(* Logix 5000 project; controller DC01 vendor 1 type 14 code 165 rev 32.12; software revision 32.04 *)

TASK MainTask (continuous, watchdog 500 ms) : MainProgram, LN01, LN02, LN03, LN04

MODULES
   Local : vendor 1 type 14 code 165 (ICP 0, rev 32.12)
      ASSY_LN01 : 1756-EN2T (ICP 1, Ethernet 192.168.1.211, rev 11.1)
         LN01_COMMS : 1756-EN2T (Ethernet 192.168.1.221, rev 11.2, Output RPI 10 ms)
            LN01 : vendor 1 type 14 code 167 (ICP 0, rev 32.1)
      ASSY_LN02 : 1756-EN2T (ICP 2, Ethernet 192.168.1.212, rev 11.1)
         LN02_COMMS : 1756-EN2T (Ethernet 192.168.1.222, rev 11.1, Output RPI 10 ms)
            LN02 : vendor 1 type 14 code 167 (ICP 0, rev 33.1)
      ASSY_LN03 : 1756-EN2T (ICP 3, Ethernet 192.168.1.213, rev 11.1)
         LN03_COMMS : 1756-EN2T (Ethernet 192.168.1.223, rev 11.1, Output RPI 10 ms)
            LN03 : vendor 1 type 14 code 167 (ICP 0, rev 33.1)
      ASSY_COMMS : 1756-EN2T (ICP 6, Ethernet 10.27.36.150, rev 11.2)
      ASSY_LN04 : 1756-EN2T (ICP 4, Ethernet 192.168.1.214, rev 11.1)
         LN04_COMMS : 1756-EN2T (Ethernet 192.168.1.224, rev 11.1, Output RPI 10 ms)
            LN04 : vendor 1 type 14 code 167 (ICP 0, rev 33.1)
END_MODULES

TYPE Barcode_SNModel :
STRUCT
   Data : STRING[5];
   Bit : BOOL[32];
END_STRUCT
END_TYPE

TYPE BARCODESCAN :
STRUCT
   RAWDATA : STRING;
   TRIGGER : BOOL;
   CLEAR : BOOL;
   SCANCOMPLETE : BOOL;
END_STRUCT
END_TYPE

TYPE Data_RECT :
STRUCT
   Volt_Out : INT;
   Amp_Out : INT;
   DC_ON : BOOL;
END_STRUCT
END_TYPE

TYPE DateTime_Type :   // Structure for the DateTime from the Controller wallclock accessed by the GSV/SSV instruction
STRUCT
   Year : DINT;
   Month : DINT;   // The month (1 - 12)
   Day : DINT;   // The day (1 - 31)
   Hour : DINT;   // hour (0 - 23)
   Minute : DINT;   // minute (0 - 59)
   Second : DINT;   // second (0 - 59)
   Microseconds : DINT;   // (0 - 999,999)
END_STRUCT
END_TYPE

TYPE DriveData :
STRUCT
   FieldAmps : REAL;
   VoltsOut : REAL;
   ArmCurrent : REAL;
   ActualSpeed : REAL;
END_STRUCT
END_TYPE

TYPE DriveDataDINT :
STRUCT
   FieldAmps : DINT;
   ArmAmps : DINT;
   OutVolts : DINT;
   Speed : DINT;
END_STRUCT
END_TYPE

TYPE Drives1079 :
STRUCT
   Drive1 : DriveData;
   Drive2 : DriveData;
   Drive3 : DriveData;
   Drive4 : DriveData;
   Drive5 : DriveData;
   Drive6 : DriveData;
END_STRUCT
END_TYPE

TYPE Drives1079DINT :
STRUCT
   Drive1 : DriveDataDINT;
   Drive2 : DriveDataDINT;
   Drive3 : DriveDataDINT;
   Drive4 : DriveDataDINT;
   Drive5 : DriveDataDINT;
   Drive6 : DriveDataDINT;
END_STRUCT
END_TYPE

TYPE Lodestar_Data_DINTS :
STRUCT
   Mode : DINT;
   State : DINT;
   AutoMan : DINT;
   Process : DINT;
   Rate : DINT;
   Fault_Code : DINT;
   Infeed_Count : DINT;
   OutFeed_Count : DINT;
   Reject_Count : DINT;
   Cycle_Count : DINT;
END_STRUCT
END_TYPE

TYPE LPNSTATUS :   // Data From SQL for Online Printing to tell what Current Model the line is in
STRUCT
   LineID : INT;   // Line Number
   Total_Run : INT;   // Total Number of Units in Current Run
   Produced : INT;   // Total Number of Units Ran in Current Run
   Left_To_Run : INT;   // Total Number of Units Left to Run in Current Run
   Model : STRING;   // Model Number of Current Run
END_STRUCT
END_TYPE

TYPE OnlinePrinitng :
STRUCT
   ENGMODEL : STRING;
   SALESMODEL : STRING;
   MODEL : STRING;
   SERIAL : STRING;
   DATA_TO_APP_READY : BOOL;
   APP_DATA_RECEIVED : BOOL;
   DATA_FROM_APP_READY : BOOL;
   LINERUNNING : BOOL;
   CLEAR : BOOL;
   BARCODEDATA : BARCODESCAN;
END_STRUCT
END_TYPE

TYPE PA_WallClock_UDDT :
STRUCT
   One_Shots : BOOL[128];
   Bool : BOOL[128];
   Real : REAL[50];
   Dbl_Int : DINT[50];
   Int : INT[50];
   Pointer1 : INT;
   Pointer2 : INT;
   Pointer3 : INT;
   Pointer4 : INT;
   Pointer5 : INT;
   Timer : TIMER[50];
   Counter : COUNTER[25];
   Control : CONTROL[16];
END_STRUCT
END_TYPE

TYPE R1_Lines_Status_to_R2 :
STRUCT
   LN02 : UDT_Line_Status_to_R2;
   LN03 : UDT_Line_Status_to_R2;
   LN04 : UDT_Line_Status_to_R2;
   LN07 : UDT_Line_Status_to_R2;
END_STRUCT
END_TYPE

TYPE R3_Ticket_Data :   // Ticket Data from LN04 Scanners
STRUCT
   Model : STRING;
   Date : STRING;
   Serial : STRING;
END_STRUCT
END_TYPE

TYPE R3_Ticket_Data2 :
STRUCT
   Model : STRING;
   Date : STRING;
   Serial : STRING;
END_STRUCT
END_TYPE

TYPE RECT_1079 :
STRUCT
   RECT1 : Data_RECT;
   RECT2 : Data_RECT;
   RECTBU : Data_RECT;
END_STRUCT
END_TYPE

TYPE STRING_12 :
STRUCT
   LEN : DINT;
   DATA : SINT[12];
END_STRUCT
END_TYPE

TYPE STRING_16 :
STRUCT
   LEN : DINT;
   DATA : SINT[16];
END_STRUCT
END_TYPE

TYPE STRING_24 :
STRUCT
   LEN : DINT;
   DATA : SINT[24];
END_STRUCT
END_TYPE

TYPE STRING_4 :
STRUCT
   LEN : DINT;
   DATA : SINT[4];
END_STRUCT
END_TYPE

TYPE STRING_40 :
STRUCT
   LEN : DINT;
   DATA : SINT[40];
END_STRUCT
END_TYPE

TYPE UDT_Current_Status :
STRUCT
   Area : STRING_12;
   Line : STRING_12;
   Shift : DINT;
   _1st_Shift_Avail : BOOL;
   _1st_Shift_Active : BOOL;
   _1st_Shift_Scheduled : BOOL;
   _2nd_Shift_Avail : BOOL;
   _2nd_Shift_Active : BOOL;
   _2nd_Shift_Scheduled : BOOL;
   _3rd_Shift_Avail : BOOL;
   _3rd_Shift_Active : BOOL;
   _3rd_Shift_Scheduled : BOOL;
   DayOfWeek : STRING_16;
   DayOfWeek_Int : DINT;
   Start_Time : STRING_16;
   End_Time : STRING_16;
   _1st_Break_Time : STRING_16;
   _1st_Break_Trigger : BOOL;
   _1st_Break_Active : BOOL;
   _1st_Break_Used : BOOL;
   Lunch_Time : STRING_16;
   Lunch_Trigger : BOOL;
   Lunch_Active : BOOL;
   Lunch_Used : BOOL;
   _2nd_Break_Time : STRING_16;
   _2nd_Break_Trigger : BOOL;
   _2nd_Break_Active : BOOL;
   _2nd_Break_Used : BOOL;
   Rotate_Active : BOOL;
   Rotate_Cmd : BOOL;   // 30 Second Downtime Event to Rotate the Crew
   Scheduled_Units : DINT;
   Line_Rate : DINT;   // Seconds to Construct a Component
   Line_Rate_SP : REAL;
   Units_Remaining : DINT;
   Units_Produced : DINT;
   Units_Scrapped : DINT;
   Units_Lossed : DINT;
   AY_Percent : REAL;
   Shift_Minutes_Remainng : DINT;
   Shift_Seconds_Remaining : DINT;
   DownTime_Code : DINT;
   Flex_Cmd : BOOL;
   Flex_Active : BOOL;
   FlexTo_Line : STRING_16;
   Flex_EndCmd : BOOL;
   Rotate_LEN : REAL;   // seconds
   Brk_LEN : REAL;   // minutes
   Lunch_LEN : REAL;   // minutes
   Break_Stop_On : BOOL;
   Break_Stop_Allowed : BOOL;
   Flex_Stop_On : BOOL;
   Flex_Stop_Allowed : BOOL;
   Rotate_Stop_On : BOOL;
   Rotate_Stop_Allowed : BOOL;
   S1_Scheduled : DINT;
   S2_Scheduled : DINT;
   S3_Scheduled : DINT;
   Shift_Scheduled : BOOL;
   Shift_Active : BOOL;
   RateToMakeSchedule : REAL;
   Theoretical_Units : DINT;
   Standard_LineRate : REAL;
   Running : BOOL;
   State : DINT;
   LineWide_Event : DINT;
   Units_Rejected : DINT;
END_STRUCT
END_TYPE

TYPE UDT_Daily_Schedule :
STRUCT
   _1st_Shift_Avail : BOOL;
   _1st_Shift_Start : STRING_16;
   _1st_Shift_End : STRING_16;
   _1st_Shift_Break1_Start : STRING_16;
   _1st_Shift_Break1_Length : DINT;   // Minutes
   _1st_Shift_Lunch_Start : STRING_16;
   _1st_Shift_Lunch_Length : DINT;   // Minutes
   _1st_Shift_Break2_Start : STRING_16;
   _1st_Shift_Break2_Length : DINT;   // Minutes
   _2nd_Shift_Avail : BOOL;
   _2nd_Shift_Start : STRING_16;
   _2nd_Shift_End : STRING_16;
   _2nd_Shift_Break1_Start : STRING_16;
   _2nd_Shift_Break1_Length : DINT;   // Minutes
   _2nd_Shift_Lunch_Start : STRING_16;
   _2nd_Shift_Lunch_Length : DINT;   // Minutes
   _2nd_Shift_Break2_Start : STRING_16;
   _2nd_Shift_Break2_Length : DINT;   // Minutes
   _3rd_Shift_Avail : BOOL;
   _3rd_Shift_Start : STRING_16;
   _3rd_Shift_End : STRING_16;
   _3rd_Shift_Break1_Start : STRING_16;
   _3rd_Shift_Break1_Length : DINT;   // Minutes
   _3rd_Shift_Lunch_Start : STRING_16;
   _3rd_Shift_Lunch_Length : DINT;   // Minutes
   _3rd_Shift_Break2_Start : STRING_16;
   _3rd_Shift_Break2_Length : DINT;   // Minutes
   Rotate_Length : DINT;   // Seconds
   Break_Stop_On : BOOL;
   Break_Stop_Allowed : BOOL;
   Flex_Stop_On : BOOL;
   Flex_Stop_Allowed : BOOL;
   Rotate_Stop_On : BOOL;
   Rotate_Stop_Allowed : BOOL;
   S1_Scheduled : DINT;
   S2_Scheduled : DINT;
   S3_Scheduled : DINT;
   RateToMakeSchedule : REAL;
END_STRUCT
END_TYPE

TYPE UDT_DateTime :
STRUCT
   Year : STRING_4;
   Month : STRING_4;
   Day : STRING_4;
   Hour : STRING_4;
   Minute : STRING_4;
   Second : STRING_4;
   MicroSecond : STRING_4;
   ForwardSlash : STRING_4;
   Colon : STRING_4;
   Period : STRING_4;
   Zero : STRING_4;
   Final : STRING_4;
   Space : STRING_4;
   Millisecond : STRING_4;
END_STRUCT
END_TYPE

TYPE UDT_Downtime_Testing :
STRUCT
   Line_Scheduled : BOOL;
   Break : BOOL;
   Set_ModelNumber : BOOL;
   Downtime_Active : BOOL;
   Shift_Reset : BOOL;
   CrateCount_Trigger : BOOL;
   Set_TAKT : BOOL;
   TAKT_Time : DINT;
   SerialNumber_Length : DINT;
   Dev : DINT;
   Current_Shift : DINT;
   OneShots : DINT;
   LineRate : REAL;
   Production_Crate_Count_TMR : TIMER;
   Set_TAKT_Delay_TMR : TIMER;
   CrateCountTrigger_TMR : TIMER;
   Sch_Production_Crate_Count_TMR : TIMER;
   SerialNumber_Generator_CNTR : COUNTER;
   Units_Produced_CNTR : COUNTER;
   Scheduled_Units_CNTR : COUNTER;
   ModelNumber : STRING;
   TempModelNumber : STRING;
   SerialNumber : STRING;
   SalesModelNumber : STRING;
   zeros_7 : STRING_12;
   zeros_6 : STRING_12;
   zeros_5 : STRING_12;
   zeros_4 : STRING_12;
   zeros_3 : STRING_4;
   zeros_2 : STRING_4;
   zeros_1 : STRING_4;
   LineID : STRING;
END_STRUCT
END_TYPE

TYPE UDT_Line_Status_to_R2 :
STRUCT
   Active_Shift : DINT;
   Count : DINT;
   Break_Active : BOOL;
   DT_Active : BOOL;
END_STRUCT
END_TYPE

TYPE UDT_R3_BlackOut :   // Defines start and stop times for R3 schedule true ups, this apples to all lines in Clyde
STRUCT
   Starthour : DINT;
   StartMinute : DINT;
   EndHour : DINT;
   EndMinute : DINT;
END_STRUCT
END_TYPE

TYPE UDT_R3_Missed_Scan :
STRUCT
   New_Serial : BOOL;
   Same_Serial_TMR : TIMER;
   Prev_Count : DINT;
   New_Serial_TMR : TIMER;
   Missed_Scan_TMR : TIMER;
   Prev_Serial : STRING;
END_STRUCT
END_TYPE

TYPE UDT_R3_Model_Information :   // Provides structure for getting information from Ignition related to Changeover information
STRUCT
   Model : STRING;
   Count : DINT;
   Order : DINT;
   SEQ_No : DINT;
   SAP_Received_QTY : DINT;
   Description : STRING;
END_STRUCT
END_TYPE

TYPE UDT_ScantoExitDatatoDC :
STRUCT
   Serial : STRING;
   Model : STRING;
   Pass : BOOL;
   Fail : BOOL;
   Location : DINT;
END_STRUCT
END_TYPE

TYPE UDT_SHIFT_FPY :   // Shift FPY FOR line 2,3,4,7
STRUCT
   Line_2_FPY : REAL;   // Line 2
   Line_3_FPY : REAL;   // Line 3
   Line_4_FPY : REAL;   // Line 4
   Line_7_FPY : REAL;   // Line 7
END_STRUCT
END_TYPE

TYPE UDT_ShiftString_Breakdown :
STRUCT
   s1StartHour : STRING_4;
   s1StartMin : STRING_4;
   s1EndHour : STRING_4;
   s1_EndMin : STRING_4;
   s2StartHour : STRING_4;
   s2StartMin : STRING_4;
   s2EndHour : STRING_4;
   s2EndMin : STRING_4;
   s3StartHour : STRING_4;
   s3StartMin : STRING_4;
   s3EndHour : STRING_4;
   s3EndMin : STRING_4;
   break1StartHour : STRING_4;
   break1StartMin : STRING_4;
   break2StartHour : STRING_4;
   break2StartMin : STRING_4;
   lunchStartHour : STRING_4;
   lunchStartMin : STRING_4;
END_STRUCT
END_TYPE

TYPE udt_SKU :
STRUCT
   Name : STRING;   // Name of product
   Diameter : REAL;   // Diameter in millimeters
   Height : REAL;   // Height in millimeters
   ID : INT;   // Product ID
   DiameterID : REAL;
   HeightID : REAL;
   Update : BOOL;
   Update_ONS : BOOL;
   Active : BOOL;
   Active_Req : BOOL;
   UpdatePB : BOOL;
   TooManyActive : BOOL;
   DestinationOut : INT;
   ActivePB : BOOL;
   BatchRequest : INT;
   BatchCount : INT;
   ASRS_Enabled : BOOL;
   DestinationIn : INT;
   ResetPB : BOOL;
   BatchComplete : BOOL;
END_STRUCT
END_TYPE

TYPE UDT_SN_Model :
STRUCT
   writeIndex : DINT;
   readIndex : DINT;
   LastReadCode : DINT;
   Serial : STRING_16;
   Model : STRING_16;
   DateTime : STRING_24;
   newData : BOOL;
END_STRUCT
END_TYPE

TYPE UDT_Visual_Inspect_Data :   // UDT from Assy lines for Scanners that track models
STRUCT
   Date : STRING;
   Unit_Status : BOOL;
   Model : STRING;
   Serial : STRING;
   Badge_ID : DINT;
   Data_Ready : BOOL;
END_STRUCT
END_TYPE

TYPE UDT_Visual_Inspect_Data2 :
STRUCT
   DATE : STRING;
   UNIT_STATUS : BOOL;
   MODEL : STRING;
   SERIAL : STRING;
   BADGE_ID : DINT;
   DATA_READY : BOOL;
END_STRUCT
END_TYPE

TYPE UDT_Weekly_Schedule :
STRUCT
   Monday : UDT_Daily_Schedule;
   Tuesday : UDT_Daily_Schedule;
   Wednesday : UDT_Daily_Schedule;
   Thursday : UDT_Daily_Schedule;
   Friday : UDT_Daily_Schedule;
   Saturday : UDT_Daily_Schedule;
   Sunday : UDT_Daily_Schedule;
END_STRUCT
END_TYPE

TYPE Visual_Inspect_Data :
STRUCT
   DATE : STRING;
   UNIT_STATUS : BOOL;
   MODEL : STRING;
   SERIAL : STRING;
   BADGE_ID : DINT;
   DATA_READY : BOOL;
END_STRUCT
END_TYPE

VAR_GLOBAL   (* controller tags *)
   Always_Off : BOOL;
   apc_debounce : TIMER := (PRE := 1100);
   apc_DT_CTR : TIMER := (PRE := 999999999);
   ASSY_COMS_com_status : DINT := 16384;   // DC01 Bldg Ethernet Communications To Data Center Status Monitor
   ay : REAL := 0.8867925;
   ay_LN01 : DINT;
   ay_LN01_REAL : REAL := 0.95028526;
   AY_LN02_REAL : REAL := 0.9279279;
   Barcode_Scan : MESSAGE;
        MessageParameters(ServiceCode := 16#004c, LocalElement := LN01_Messages_Barcode_SNModel, ...)
   brentest : BOOL;
   brentest2 : BOOL := 1;
   Brian_Test : BOOL;
   ChangeWEM15TO12 : BOOL := 1;
   clock_current_string : STRING[13] := ([0] := '2023', [1] := '5', [2] := '8', [3] := '7', [4] := '52', [5] := '42');
   Clock_Min_Pulse : BOOL;
   Clock_Set_Routine : PA_WallClock_UDDT := (Bool[20] := 1, Dbl_Int[40] := 2023, Dbl_Int[41] := 5, Dbl_Int[42] := 8, Dbl_Int[43] := 7, Dbl_Int[44] := 52, Dbl_Int[45] := 43, Dbl_Int[46] := 547971, Timer[0].PRE := 500, Timer[8].EN := 1, Timer[8].TT := 1, Timer[9].ACC := 100, Timer[9].EN := 1, Timer[9].DN := 1);
   covid19 : BOOL;
   CurrentSchedule : UDT_ShiftString_Breakdown := (s1StartHour := '20', s1StartMin := '3-', s1EndHour := '20', s1_EndMin := '3-', s2StartHour := '20', s2StartMin := '3-', s2EndHour := '20', s2EndMin := '3-', s3StartHour := '20', s3StartMin := '3-', s3EndHour := '20', s3EndMin := '3-');
   DateTime_Update : BOOL;
   DayOfWeek : DINT;
   DC01_to_LN04_Data : DINT[26] := ([1] := 201);
   DC1_clock_sync : DINT[10] := ([0] := 2023, [1] := 5, [2] := 8, [3] := 7, [4] := 52, [5] := 43);
   DC1_OPCFault : BOOL := 1;
   DC1_OPCWatchDog : BOOL := 1;
   DC1_to_LN01_Messages : DINT[20] := ([0] := 1, [2] := 1, [3] := 1240, [4] := 598, [5] := 7, [6] := 5, [7] := 15, [8] := 28, [9] := 15, [10] := 35, [11] := 23, [12] := 58, [14] := 5, [15] := 6, [16] := 58, [17] := 33900, [19] := 1);
        [10]   // CURRENT SCHEDULE SHIFT 2 START MINUTE
        [11]   // CURRENT SCHEDULE SHIFT 2 END HOUR
        [12]   // CURRENT SCHEDULE SHIFT 2 END MINUTE
        [13]   // CURRENT SCHEDULE SHIFT 3 START HOUR
        [14]   // CURRENT SCHEDULE SHIFT 3 START MINUTE
        [15]   // CURRENT SCHEDULE SHIFT 3 END HOUR
        [16]   // CURRENT SCHEDULE SHIFT 3 END MINUTE
        [17]   // CURRENT SCHEDULE AVAILABLE SECONDS
        [19].0   // SHIFT SCHEDULED
        [19].1   // OPC COMMS OKAY
        [2]   // ACTIVE SHIFT
        [3]   // SCHEDULED UNITS
        [5]   // CURRENT SCHEDULE SHIFT 1 START HOUR
        [6]   // CURRENT SCHEDULE SHIFT 1 START MINUTE
        [7]   // CURRENT SCHEDULE SHIFT 1 END HOUR
        [8]   // CURRENT SCHEDULE SHIFT 1 END MINUTE
        [9]   // CURRENT SCHEDULE SHIFT 2 START HOUR
        [0]   // DC01 STATUS TO ASSY LN01
        [0].0   // DC01 Ethernet Building Network Comms Good to Line 1 Processor
   DC1_to_LN02_Messages : DINT[20] := ([0] := 1, [2] := 1, [3] := 1240, [4] := 598, [5] := 7, [6] := 5, [7] := 15, [8] := 28, [9] := 15, [10] := 35, [11] := 23, [12] := 58, [14] := 5, [15] := 6, [16] := 58, [17] := 33900, [19] := 1);
        [10]   // CURRENT SCHEDULE SHIFT 2 START MINUTE
        [11]   // CURRENT SCHEDULE SHIFT 2 END HOUR
        [12]   // CURRENT SCHEDULE SHIFT 2 END MINUTE
        [13]   // CURRENT SCHEDULE SHIFT 3 START HOUR
        [14]   // CURRENT SCHEDULE SHIFT 3 START MINUTE
        [15]   // CURRENT SCHEDULE SHIFT 3 END HOUR
        [16]   // CURRENT SCHEDULE SHIFT 3 END MINUTE
        [17]   // CURRENT SCHEDULE AVAILABLE SECONDS
        [19].0   // SHIFT SCHEDULED
        [19].1   // OPC COMMS OKAY
        [2]   // ACTIVE SHIFT
        [3]   // SCHEDULED UNITS
        [5]   // CURRENT SCHEDULE SHIFT 1 START HOUR
        [6]   // CURRENT SCHEDULE SHIFT 1 START MINUTE
        [7]   // CURRENT SCHEDULE SHIFT 1 END HOUR
        [8]   // CURRENT SCHEDULE SHIFT 1 END MINUTE
        [9]   // CURRENT SCHEDULE SHIFT 2 START HOUR
        [0]   // DC01 STATUS TO ASSY LN02
        [0].0   // DC01 Ethernet Building Network Comms Good to Line 2 Processor
   DC1_to_LN03_Messages : DINT[20] := ([0] := 1, [2] := 1, [3] := 700, [4] := 337, [5] := 7, [6] := 5, [7] := 15, [8] := 28, [9] := 15, [10] := 35, [11] := 23, [12] := 58, [14] := 5, [15] := 6, [16] := 58, [17] := 33900, [19] := 1);
        [10]   // CURRENT SCHEDULE SHIFT 2 START MINUTE
        [11]   // CURRENT SCHEDULE SHIFT 2 END HOUR
        [12]   // CURRENT SCHEDULE SHIFT 2 END MINUTE
        [13]   // CURRENT SCHEDULE SHIFT 3 START HOUR
        [14]   // CURRENT SCHEDULE SHIFT 3 START MINUTE
        [15]   // CURRENT SCHEDULE SHIFT 3 END HOUR
        [16]   // CURRENT SCHEDULE SHIFT 3 END MINUTE
        [17]   // CURRENT SCHEDULE AVAILABLE SECONDS
        [19].0   // SHIFT SCHEDULED
        [19].1   // OPC COMMS OKAY
        [2]   // ACTIVE SHIFT
        [3]   // SCHEDULED UNITS
        [5]   // CURRENT SCHEDULE SHIFT 1 START HOUR
        [6]   // CURRENT SCHEDULE SHIFT 1 START MINUTE
        [7]   // CURRENT SCHEDULE SHIFT 1 END HOUR
        [8]   // CURRENT SCHEDULE SHIFT 1 END MINUTE
        [9]   // CURRENT SCHEDULE SHIFT 2 START HOUR
        [0]   // DC01 STATUS TO ASSY LN03
        [0].0   // DC01 Ethernet Building Network Comms Good to Line 3 Processor
   DC1_to_LN04_Messages : DINT[20] := ([0] := 1, [2] := 1, [3] := 425, [4] := 205, [5] := 7, [6] := 5, [7] := 15, [8] := 28, [9] := 15, [10] := 35, [11] := 23, [12] := 58, [14] := 5, [15] := 6, [16] := 58, [17] := 33900, [19] := 1);
        [10]   // CURRENT SCHEDULE SHIFT 2 START MINUTE
        [11]   // CURRENT SCHEDULE SHIFT 2 END HOUR
        [12]   // CURRENT SCHEDULE SHIFT 2 END MINUTE
        [13]   // CURRENT SCHEDULE SHIFT 3 START HOUR
        [14]   // CURRENT SCHEDULE SHIFT 3 START MINUTE
        [15]   // CURRENT SCHEDULE SHIFT 3 END HOUR
        [16]   // CURRENT SCHEDULE SHIFT 3 END MINUTE
        [17]   // CURRENT SCHEDULE AVAILABLE SECONDS
        [19].0   // SHIFT SCHEDULED
        [19].1   // OPC COMMS OKAY
        [2]   // ACTIVE SHIFT
        [3]   // SCHEDULED UNITS
        [5]   // CURRENT SCHEDULE SHIFT 1 START HOUR
        [6]   // CURRENT SCHEDULE SHIFT 1 START MINUTE
        [7]   // CURRENT SCHEDULE SHIFT 1 END HOUR
        [8]   // CURRENT SCHEDULE SHIFT 1 END MINUTE
        [9]   // CURRENT SCHEDULE SHIFT 2 START HOUR
        [0]   // DC01 STATUS TO ASSY LN04
        [0].0   // DC01 Ethernet Building Network Comms Good to Line 4 Processor
        [4]   // CURRENT SCHEDULED UNITS
   Delay_TMR_APC : TIMER := (PRE := 2000);
   Disable : DINT;
   DT_Minutes : REAL := 0.38376668;
   Elongation_Timer : TIMER[5] := ([0].PRE := 2000, [1].PRE := 2000, [2].PRE := 2000, [3].PRE := 2000, [4].PRE := 2000);
   ENET_COMMS_OK : BOOL := 1;   // DC01 Ethernet Building Network Comms Good
   fifi_unload : DINT := 1;
   IGN_DateTime_Record_Current : STRING := '2019,11,26,10:56:00';
   IGN_Day : DINT := 8;
   IGN_DayPrev : DINT := 8;
   IGN_DayString : STRING := '8';
   IGN_Hour : DINT := 7;
   IGN_HourString : STRING := '7';
   IGN_Minute : DINT := 52;
   IGN_MinuteString : STRING := '52';
   IGN_Month : DINT := 5;
   IGN_MonthString : STRING := '5';
   IGN_Second : DINT := 44;
   IGN_SecondString : STRING := '44';
   IGN_Year : DINT := 2023;
   IGN_YearString : STRING := '2023';
   L1_30min_Break_Timer : TIMER;
   L2_30min_Break_Timer : TIMER := (PRE := 1800000);
   L2_Blocked_On : BOOL := 1;
   L3_30min_Break_Timer : TIMER := (PRE := 1800000);
   L4_30min_Break_Timer : TIMER := (PRE := 1800000);
   Latch_off : BOOL;
   Latch_off1 : BOOL;
   LN01_1st_Station_Break_Code : DINT := 16;
   LN01_Additional_Break_Limit_Mins : DINT := 570;
   LN01_assist1 : DINT;
   LN01_assist2 : DINT;
   LN01_assist3 : DINT;
   LN01_assist4 : DINT;
   LN01_Assist_CT : DINT;
   LN01_Assist_Record : STRING := '02EDM-35';
   Ln01_Assist_Tag : STRING := 'ASSIST';
   LN01_Assist_Tags : STRING[5];
   LN01_Boxing_MNT : DINT;
   LN01_Cabinet_Messages : DINT[250];
   LN01_CabinetLine_MSG : MESSAGE;
   LN01_Ceran_MNT : DINT;
   LN01_Console_Messages : DINT[250] := ([9] := 1);
   LN01_Console_MNT : DINT;
   LN01_ConsoleLine_MSG : MESSAGE;
   LN01_Cooktop_MNT : DINT;
   LN01_Crating_Messages : DINT[250] := ([41] := 1);
   LN01_CratingLine_MSG : MESSAGE;
        MessageParameters(ServiceCode := 16#004c, LocalElement := LN01_Crating_Messages[0], ...)
   LN01_Current_Shift_Duration_Mins : DINT := 510;
   LN01_Current_Shift_Duration_wBreaks_Mins : DINT := 460;
   LN01_DataFromDC1 : DINT[20] := ([5] := 20, [6] := 3, [7] := 20, [8] := 3, [9] := 20, [10] := 3, [11] := 20, [12] := 3, [13] := 20, [14] := 3, [15] := 20, [16] := 3);
   LN01_DataFromDC3 : DINT[20] := ([5] := 6, [6] := 33, [7] := 15, [9] := 15, [10] := 3, [11] := 21, [12] := 45, [13] := 21, [14] := 48, [15] := 6, [16] := 15, [19] := 1);
   LN01_DC_Controlled_Theoretical_Units : BOOL := 1;
   LN01_Door_MNT : DINT;
   LN01_FinalHiPot_Messages : DINT[200] := ([9] := 1);
   LN01_FinalHiPot_MSG : MESSAGE;
        MessageParameters(ServiceCode := 16#004c, LocalElement := LN01_FinalHiPot_Messages[0], ...)
   LN01_FPY : DINT := 99;
   LN01_FrontFrame_MNT : DINT;
   LN01_Ignition_NewSNModel : BOOL[32];
   LN01_Ignition_SNModelMSG : STRING[5] := ([0] := 'WFE505W0HB 5', [1] := 'RC1827187');
   LN01_InitHiPot_Messages : DINT[200] := ([9] := 1);
   LN01_InitHiPot_MSG : MESSAGE;
        MessageParameters(ServiceCode := 16#004c, LocalElement := LN01_InitHiPot_Messages[0], ...)
   LN01_Last_Message : STRING := 'SHIFT AY ==> 97.69 %';
   LN01_MachineOverAll_MNT : DINT;
   LN01_Main_Messages : DINT[250] := ([4] := 548, [9] := 1, [14] := 10537, [15] := 99, [16] := 17, [17] := 1, [18] := 150, [19] := -7);
   LN01_MainBack_MNT : DINT;
   LN01_MainLine_MSG_Out : MESSAGE;
        MessageParameters(ServiceCode := 16#004d, LocalElement := DC1_to_LN01_Messages[0], ...)
   LN01_Match : DINT;
   LN01_Match_No_Error : DINT;
   LN01_Message_Change : BOOL := 1;
   LN01_Messages_Barcode_SNModel : Barcode_SNModel := (Data[0] := 'WFE505W0HB 5', Data[1] := 'RC1827187');
   LN01_ML_Message : STRING := 'SHIFT AY ==> 97.69 %';
   LN01_MLC_Downtime : BOOL;
   LN01_OT_Shift_Break_In_Minutes : DINT := 60;
   LN01_OvenCavity_MNT : DINT;
   LN01_Planetary_Messages : DINT[250];
   LN01_PlanetaryLine_MSG : MESSAGE;
        MessageParameters(ServiceCode := 16#004c, LocalElement := LN01_Planetary_Messages[0], ...)
   LN01_Progress_Messages : DINT[250];
   LN01_ProgressLine_MSG : MESSAGE;
        MessageParameters(ServiceCode := 16#004c, LocalElement := LN01_Progress_Messages[0], ...)
   LN01_RepairBay_Messages : DINT[200] := ([9] := 1);
   LN01_RepairBayLine_MSG : MESSAGE;
        MessageParameters(ServiceCode := 16#004c, LocalElement := LN01_RepairBay_Messages[0], ...)
   LN01_Schedule : UDT_Current_Status := (Line := 'LN01', Shift := 1, _1st_Shift_Avail := 1, _1st_Shift_Active := 1, _1st_Shift_Scheduled := 1, _2nd_Shift_Scheduled := 1, DayOfWeek := 'Mon', DayOfWeek_Int := 1, Start_Time := '2023-05-05 16:45', End_Time := '2023-05-06 01:15', Scheduled_Units := 1240, Units_Remaining := 990, Units_Produced := 548, Units_Lossed := 65, AY_Percent := 95.02853, Shift_Scheduled := 1, Shift_Active := 1, Theoretical_Units := 597, Running := 1, State := 3, Units_Rejected := 17);
   LN01_Schedule_Cycle_Time : TIMER := (PRE := 22);
   LN01_Schedule_Cycle_Timer : TIMER := (PRE := 22494, ACC := 16055, EN := 1, TT := 1);
   LN01_Schedule_Max_Break_Duration : DINT := 50;
   LN01_Schedule_Max_Break_Timer : TIMER := (PRE := 3000000, ACC := 3000000);
   LN01_Schedule_Tag : STRING := 'SCHED';
   LN01_Schedule_TAKT : REAL := 22258.064;
   LN01_Scheduled_Units_Buffer : DINT;
   LN01_ScheduleUnits_Produced_from_line : DINT := 49339;
   LN01_SidePanel_MNT : DINT;
   LN01_SidePanels_MNT : DINT;
   LN01_SNModel_Array : UDT_SN_Model[50] := ([0].LastReadCode := 1, [0].Serial := 'CA0807380', [0].Model := 'WTW4816FW2', [0].DateTime := '2/25/2021 12:28:40.38102', [1].writeIndex := 1, [1].readIndex := 1, [1].LastReadCode := 1, [1].Serial := 'CA0807381', [1].Model := 'WTW4816FW2', [1].DateTime := '2/25/2021 12:28:52.55128', [2].writeIndex := 2, [2].readIndex := 2, [2].LastReadCode := 1, [2].Serial := 'CA0807382', [2].Model := 'WTW4816FW2', [2].DateTime := '2/25/2021 12:29:03.43928', [3].writeIndex := 3, [3].readIndex := 3, [3].LastReadCode := 1, [3].Serial := 'CA0807383', [3].Model := 'WTW4816FW2', [3].DateTime := '2/25/2021 12:29:14.30134', [4].writeIndex := 4, [4].readIndex := 4, [4].LastReadCode := 1, [4].Serial := 'CA0807384', [4].Model := 'WTW4816FW2', [4].DateTime := '2/25/2021 12:29:24.42454', [5].writeIndex := 5, [5].readIndex := 5, [5].LastReadCode := 1, [5].Serial := 'CA0807385', [5].Model := 'WTW4816FW2', [5].DateTime := '2/25/2021 12:29:35.71676', [6].writeIndex := 6, [6].readIndex := 6, [6].LastReadCode := 1, [6].Serial := 'CA0807386', [6].Model := 'WTW4816FW2', [6].DateTime := '2/25/2021 12:29:46.65221', [7].writeIndex := 7, [7].readIndex := 7, [7].LastReadCode := 1, [7].Serial := 'CA0807387', [7].Model := 'WTW4816FW2', [7].DateTime := '2/25/2021 12:29:57.14076', [8].writeIndex := 8, [8].readIndex := 8, [8].LastReadCode := 1, [8].Serial := 'CA0807388', [8].Model := 'WTW4816FW2', [8].DateTime := '2/25/2021 12:30:38.78655', [9].writeIndex := 10, [9].readIndex := 9, [9].LastReadCode := 1, [9].Serial := 'CA0807389', [9].Model := 'WTW4816FW2', [9].DateTime := '2/25/2021 12:30:51.72217', [10].writeIndex := 10, [10].readIndex := 10,
        [10].LastReadCode := 1, [10].Serial := 'CA0807390', [10].Model := 'WTW4816FW2', [10].DateTime := '2/25/2021 12:31:01.80920', [11].writeIndex := 11, [11].readIndex := 11, [11].LastReadCode := 1, [11].Serial := 'CA0807391', [11].Model := 'WTW4816FW2', [11].DateTime := '2/25/2021 12:31:11.91238', [12].writeIndex := 12, [12].readIndex := 12, [12].LastReadCode := 1, [12].Serial := 'CA0807392', [12].Model := 'WTW4816FW2', [12].DateTime := '2/25/2021 12:31:24.82835', [13].writeIndex := 13, [13].readIndex := 13, [13].LastReadCode := 1, [13].Serial := 'CA0807393', [13].Model := 'WTW4816FW2', [13].DateTime := '2/25/2021 12:31:33.33885', [14].writeIndex := 14, [14].readIndex := 14, [14].LastReadCode := 1, [14].Serial := 'CA0807394', [14].Model := 'WTW4816FW2', [14].DateTime := '2/25/2021 12:31:44.26004', [15].writeIndex := 15, [15].readIndex := 15, [15].LastReadCode := 1, [15].Serial := 'CA0807395', [15].Model := 'WTW4816FW2', [15].DateTime := '2/25/2021 12:31:55.17391', [16].writeIndex := 16, [16].readIndex := 16, [16].LastReadCode := 1, [16].Serial := 'CA0807396', [16].Model := 'WTW4816FW2', [16].DateTime := '2/25/2021 12:32:06.90771', [17].writeIndex := 17, [17].readIndex := 17, [17].LastReadCode := 1, [17].Serial := 'CA0807397', [17].Model := 'WTW4816FW2', [17].DateTime := '2/25/2021 12:32:16.96281', [18].writeIndex := 18, [18].readIndex := 18, [18].LastReadCode := 1, [18].Serial := 'CA0807398', [18].Model := 'WTW4816FW2', [18].DateTime := '2/25/2021 12:32:27.92434', [19].writeIndex := 19, [19].readIndex := 19, [19].LastReadCode := 1, [19].Serial := 'CA0807399', [19].Model := 'WTW4816FW2', [19].DateTime := '2/25/2021 12:32:38.40881', [20].writeIndex := 20, [20].readIndex := 20,
        [20].LastReadCode := 1, [20].Serial := 'CA0807400', [20].Model := 'WTW4816FW2', [20].DateTime := '2/25/2021 12:32:49.30917', [21].writeIndex := 21, [21].readIndex := 21, [21].LastReadCode := 1, [21].Serial := 'CA0807401', [21].Model := 'WTW4816FW2', [21].DateTime := '2/25/2021 12:33:00.28133', [22].writeIndex := 22, [22].readIndex := 22, [22].LastReadCode := 1, [22].Serial := 'CA0807402', [22].Model := 'WTW4816FW2', [22].DateTime := '2/25/2021 12:33:35.38591', [23].writeIndex := 23, [23].readIndex := 23, [23].LastReadCode := 1, [23].Serial := 'CA0807403', [23].Model := 'WTW4816FW2', [23].DateTime := '2/25/2021 12:33:45.88840', [24].writeIndex := 24, [24].readIndex := 24, [24].LastReadCode := 1, [24].Serial := 'CA0807404', [24].Model := 'WTW4816FW2', [24].DateTime := '2/25/2021 12:33:56.85644', [25].writeIndex := 25, [25].readIndex := 25, [25].LastReadCode := 1, [25].Serial := 'CA0807405', [25].Model := 'WTW4816FW2', [25].DateTime := '2/25/2021 12:34:07.73473', [26].writeIndex := 26, [26].readIndex := 26, [26].LastReadCode := 1, [26].Serial := 'CA0807406', [26].Model := 'WTW4816FW2', [26].DateTime := '2/25/2021 12:34:18.63707', [27].writeIndex := 27, [27].readIndex := 27, [27].LastReadCode := 1, [27].Serial := 'CA0807407', [27].Model := 'WTW4816FW2', [27].DateTime := '2/25/2021 12:34:29.95757', [28].writeIndex := 28, [28].readIndex := 28, [28].LastReadCode := 1, [28].Serial := 'CA0807408', [28].Model := 'WTW4816FW2', [28].DateTime := '2/25/2021 12:34:41.36491', [29].writeIndex := 29, [29].readIndex := 29, [29].LastReadCode := 1, [29].Serial := 'CA0807409', [29].Model := 'WTW4816FW2', [29].DateTime := '2/25/2021 12:34:52.31039', [30].writeIndex := 30, [30].readIndex := 30,
        [30].LastReadCode := 1, [30].Serial := 'CA0807410', [30].Model := 'WTW4816FW2', [30].DateTime := '2/25/2021 12:35:05.61831', [31].writeIndex := 31, [31].readIndex := 31, [31].LastReadCode := 1, [31].Serial := 'CA0807411', [31].Model := 'WTW4816FW2', [31].DateTime := '2/25/2021 12:35:14.80057', [32].writeIndex := 32, [32].readIndex := 32, [32].LastReadCode := 1, [32].Serial := 'CA0807412', [32].Model := 'WTW4816FW2', [32].DateTime := '2/25/2021 12:35:24.99536', [33].writeIndex := 33, [33].readIndex := 33, [33].LastReadCode := 1, [33].Serial := 'CA0807413', [33].Model := 'WTW4816FW2', [33].DateTime := '2/25/2021 12:35:35.89756', [34].writeIndex := 34, [34].readIndex := 34, [34].LastReadCode := 1, [34].Serial := 'CA0807414', [34].Model := 'WTW4816FW2', [34].DateTime := '2/25/2021 12:35:49.25334', [35].writeIndex := 35, [35].readIndex := 35, [35].LastReadCode := 1, [35].Serial := 'CA0807415', [35].Model := 'WTW4816FW2', [35].DateTime := '2/25/2021 12:35:57.77427', [36].writeIndex := 36, [36].readIndex := 36, [36].LastReadCode := 1, [36].Serial := 'CA0807416', [36].Model := 'WTW4816FW2', [36].DateTime := '2/25/2021 12:36:08.66572', [37].writeIndex := 37, [37].readIndex := 37, [37].LastReadCode := 1, [37].Serial := 'CA0807417', [37].Model := 'WTW4816FW2', [37].DateTime := '2/25/2021 12:36:19.57452', [38].writeIndex := 38, [38].readIndex := 38, [38].LastReadCode := 1, [38].Serial := 'CA0807418', [38].Model := 'WTW4816FW2', [38].DateTime := '2/25/2021 12:36:30.10790', [39].writeIndex := 39, [39].readIndex := 39, [39].LastReadCode := 1, [39].Serial := 'CA0807419', [39].Model := 'WTW4816FW2', [39].DateTime := '2/25/2021 12:36:40.99675', [40].writeIndex := 40, [40].readIndex := 40,
        [40].LastReadCode := 1, [40].Serial := 'CA0807420', [40].Model := 'WTW4816FW2', [40].DateTime := '2/25/2021 12:36:51.92086', [41].writeIndex := 41, [41].readIndex := 41, [41].LastReadCode := 1, [41].Serial := 'CA0807371', [41].Model := 'WTW4816FW2', [41].DateTime := '2/25/2021 12:27:03.39945', [42].writeIndex := 42, [42].readIndex := 42, [42].LastReadCode := 1, [42].Serial := 'CA0807372', [42].Model := 'WTW4816FW2', [42].DateTime := '2/25/2021 12:27:14.31229', [43].writeIndex := 43, [43].readIndex := 43, [43].LastReadCode := 1, [43].Serial := 'CA0807373', [43].Model := 'WTW4816FW2', [43].DateTime := '2/25/2021 12:27:25.22997', [44].writeIndex := 44, [44].readIndex := 44, [44].LastReadCode := 1, [44].Serial := 'CA0807374', [44].Model := 'WTW4816FW2', [44].DateTime := '2/25/2021 12:27:36.12574', [45].writeIndex := 45, [45].readIndex := 45, [45].LastReadCode := 1, [45].Serial := 'CA0807375', [45].Model := 'WTW4816FW2', [45].DateTime := '2/25/2021 12:27:46.64041', [46].writeIndex := 46, [46].readIndex := 46, [46].LastReadCode := 1, [46].Serial := 'CA0807376', [46].Model := 'WTW4816FW2', [46].DateTime := '2/25/2021 12:27:57.56194', [47].writeIndex := 47, [47].readIndex := 47, [47].LastReadCode := 1, [47].Serial := 'CA0807377', [47].Model := 'WTW4816FW2', [47].DateTime := '2/25/2021 12:28:08.50169', [48].writeIndex := 48, [48].readIndex := 48, [48].LastReadCode := 1, [48].Serial := 'CA0807378', [48].Model := 'WTW4816FW2', [48].DateTime := '2/25/2021 12:28:19.39640', [49].writeIndex := 49, [49].readIndex := 49, [49].LastReadCode := 1, [49].Serial := 'CA0807379', [49].Model := 'WTW4816FW2', [49].DateTime := '2/25/2021 12:28:30.29576');
   LN01_SNModel_CurrentRead : UDT_SN_Model := (writeIndex := 38, readIndex := 38, Serial := 'CA0807418', Model := 'WTW4816FW2', DateTime := '2/25/2021 12:36:30.10790');
   LN01_SNModel_STR40 : STRING_40[10] := ([0] := 'CA0807420', [1] := 'WTW4816FW2', [2] := '2/25/2021 12:36:55.546816');
   LN01_SpinWelder_Messages : DINT[200] := ([9] := 1);
   LN01_SpinWelder_MSG : MESSAGE;
        MessageParameters(ServiceCode := 16#004c, LocalElement := LN01_SpinWelder_Messages[0], ...)
   LN01_Standard_Shift_Break_In_Minutes : DINT := 50;
   LN01_StorageDrawer_MNT : DINT;
   LN01_Test_MNT : DINT;
   LN01_Theoretical_Units_Counter : COUNTER := (PRE := 999999, ACC := 960);
   LN01_Theoretical_Units_Counter_ONS : BOOL;
   LN01_Toggle_CountSource : BOOL := 1;
   LN01_Top_Messages : DINT[250] := ([9] := 1);
   LN01_TopLine_MSG : MESSAGE;
        MessageParameters(ServiceCode := 16#004c, LocalElement := LN01_Top_Messages[0], ...)
   LN01_Tub_Messages : DINT[250] := ([9] := 1);
   LN01_TubLine_MSG : MESSAGE;
        MessageParameters(ServiceCode := 16#004c, LocalElement := LN01_Tub_Messages[0], ...)
   LN01_Units_for_repair : DINT := 99;
   LN01_WaterFill_Messages : DINT[200] := ([9] := 1);
   LN01_WaterFill_MSG : MESSAGE;
        MessageParameters(ServiceCode := 16#004c, LocalElement := LN01_WaterFill_Messages[0], ...)
   LN01_Weekly_Schedule : UDT_Weekly_Schedule := (Monday._1st_Shift_Avail := 1, Monday._1st_Shift_Start := '2023-05-08 05:00', Monday._1st_Shift_End := '2023-05-08 13:30', Monday._2nd_Shift_Avail := 1, Monday._2nd_Shift_Start := '2023-05-08 16:45', Monday._2nd_Shift_End := '2023-05-09 01:15', Monday._3rd_Shift_Start := '2023-05-08 04:50', Monday._3rd_Shift_End := '2023-05-08 04:55', Monday.S1_Scheduled := 1240, Monday.S2_Scheduled := 1240, Tuesday._1st_Shift_Avail := 1, Tuesday._1st_Shift_Start := '2023-05-09 05:00', Tuesday._1st_Shift_End := '2023-05-09 15:30', Tuesday._2nd_Shift_Avail := 1, Tuesday._2nd_Shift_Start := '2023-05-09 16:45', Tuesday._2nd_Shift_End := '2023-05-10 03:15', Tuesday._3rd_Shift_Start := '2023-05-09 04:50', Tuesday._3rd_Shift_End := '2023-05-09 04:55', Tuesday.S1_Scheduled := 1537, Tuesday.S2_Scheduled := 1537, Wednesday._1st_Shift_Avail := 1, Wednesday._1st_Shift_Start := '2023-05-10 05:00', Wednesday._1st_Shift_End := '2023-05-10 15:30', Wednesday._2nd_Shift_Avail := 1, Wednesday._2nd_Shift_Start := '2023-05-10 16:45', Wednesday._2nd_Shift_End := '2023-05-11 03:15', Wednesday._3rd_Shift_Start := '2023-05-10 04:50', Wednesday._3rd_Shift_End := '2023-05-10 04:55', Wednesday.S1_Scheduled := 1537, Wednesday.S2_Scheduled := 1537, Thursday._1st_Shift_Avail := 1, Thursday._1st_Shift_Start := '2023-05-11 05:00', Thursday._1st_Shift_End := '2023-05-11 13:30', Thursday._2nd_Shift_Avail := 1, Thursday._2nd_Shift_Start := '2023-05-11 16:45', Thursday._2nd_Shift_End := '2023-05-12 01:15', Thursday._3rd_Shift_Start := '2023-05-11 04:50', Thursday._3rd_Shift_End := '2023-05-11 04:55', Thursday.S1_Scheduled := 1240, Thursday.S2_Scheduled := 1240, Friday._1st_Shift_Avail := 1, Friday._1st_Shift_Start := '2023-05-12 05:00', Friday._1st_Shift_End := '2023-05-12 13:30', Friday._2nd_Shift_Avail := 1, Friday._2nd_Shift_Start := '2023-05-12 16:45', Friday._2nd_Shift_End := '2023-05-13 01:15', Friday._3rd_Shift_Start := '2023-05-12 04:50', Friday._3rd_Shift_End := '2023-05-12 04:55', Friday.S1_Scheduled := 1240, Friday.S2_Scheduled := 1240, Saturday._1st_Shift_Start := '2023-05-13 05:00', Saturday._1st_Shift_End := '2023-05-13 13:30', Saturday._2nd_Shift_Start := '2023-05-13 16:45', Saturday._2nd_Shift_End := '2023-05-14 01:15', Saturday._3rd_Shift_Start := '2023-05-13 04:50', Saturday._3rd_Shift_End := '2023-05-13 04:55', Sunday._1st_Shift_Start := '2023-05-14 05:00', Sunday._1st_Shift_End := '2023-05-14 13:30', Sunday._2nd_Shift_Start := '2023-05-14 16:45', Sunday._2nd_Shift_End := '2023-05-15 01:15',
        Sunday._3rd_Shift_Start := '2023-05-14 04:50', Sunday._3rd_Shift_End := '2023-05-14 04:55');
   LN01_Wiring_MNT : DINT;
   LN01ECM02 : DINT;
   LN01ECM03 : DINT;
   LN01ECM04 : DINT;
   LN01ECM05 : DINT;
   LN01EDM04 : DINT;
   LN01EDM06 : DINT;
   LN01EDM07 : DINT;
   LN01EDM08 : DINT;
   LN01EEM01 : DINT;
   LN01EEM02 : DINT;
   LN01EEM03 : DINT;
   LN01EES01 : DINT;
   LN01EES02 : DINT;
   LN01EES03 : DINT;
   LN01EES04 : DINT;
   LN01EFS04 : DINT;
   LN01EFS05 : DINT;
   LN01EGM04 : DINT;
   LN01EHM01 : DINT;
   LN01EHM02 : DINT;
   LN01EHM03 : DINT;
   LN01EHM04 : DINT;
   LN01EHM05 : DINT;
   LN01EHM06 : DINT;
   LN01EHM07 : DINT;
   LN01EHM08 : DINT;
   LN01EJM02 : DINT;
   LN01EJM03 : DINT;
   LN01EKM01 : DINT;
   LN01EKM02 : DINT;
   LN01EKM03 : DINT;
   LN01ELM01 : DINT;
   LN01ELM02 : DINT;
   LN01ELM03 : DINT;
   LN01ELM04 : DINT;
   LN01ELM05 : DINT;
   LN01EMM01 : DINT;
   LN01EMM02 : DINT;
   LN01EMM03 : DINT;
   LN01NAS01 : DINT;
   LN01NAS02 : DINT;
   LN01NAS03 : DINT;
   LN01NBS02 : DINT;
   LN01SAS03 : DINT;
   LN01SBS01 : DINT;
   LN01SBS03 : DINT;
   LN01SFS03 : DINT;
   LN01SKS05 : DINT;
   LN01WAM01 : DINT;
   LN01WBM01 : DINT;
   LN01WBM02 : DINT;
   LN01WBM03 : DINT;
   LN01WBM04 : DINT;
   LN01WCM01 : DINT;
   LN01WCM02 : DINT;
   LN01WCM03 : DINT;
   LN01WCM04 : DINT;
   LN01WCM05 : DINT;
   LN01WCM06 : DINT;
   LN01WDM01 : DINT;
   LN01WDM02 : DINT;
   LN01WDM03 : DINT;
   LN01WDM04 : DINT;
   LN01WDM05 : DINT;
   LN01WFS01 : DINT;
   LN01WFS02 : DINT;
   LN01WGM01 : DINT;
   LN01WGM02 : DINT;
   LN01WGM03 : DINT;
   LN01WGM04 : DINT;
   LN01WGM05 : DINT;
   LN01WHM05 : DINT;
   LN01WHM08 : DINT;
   LN01WJS01 : DINT;
   LN01WJS02 : DINT;
   LN01WJS03 : DINT;
   LN01WKS01 : DINT;
   LN01WKS02 : DINT;
   LN01WKS03 : DINT;
   LN01WKS04 : DINT;
   LN01WLM06 : DINT;
   LN01WLM07 : DINT;
   LN01WMM02 : DINT;
   LN01ZMN01 : DINT := 16;
   LN01ZMN02 : DINT;
   LN01ZMN03 : DINT;
   LN01ZMN04 : DINT;
   LN01ZMS01 : DINT := 16;
   LN01ZMS02 : DINT;
   LN01ZMS03 : DINT;
   LN01ZMS04 : DINT;
   LN02_1st_Station_Break_Code : DINT := 16;
   LN02_Additional_Break_Limit_Mins : DINT := 570;
   LN02_assist1 : DINT;
   LN02_assist2 : DINT;
   LN02_assist3 : DINT;
   LN02_assist4 : DINT;
   LN02_Assist_CT : DINT;
   LN02_Assist_Record : STRING := '02EDM-35';
   LN02_Assist_Tag : STRING := 'ASSIST';
   LN02_Assist_Tags : STRING[5];
   LN02_Boxing_MNT : DINT;
   LN02_Ceran_MNT : DINT;
   LN02_Console_MNT : DINT;
   LN02_Cooktop_MNT : DINT;
   LN02_Current_Shift_Duration_Mins : DINT := 510;
   LN02_Current_Shift_Duration_wBreaks_Mins : DINT := 460;
   LN02_DataFromDC1 : DINT[20] := ([5] := 20, [6] := 3, [7] := 20, [8] := 3, [9] := 20, [10] := 3, [11] := 20, [12] := 3, [13] := 20, [14] := 3, [15] := 20, [16] := 3);
   LN02_DataFromDC3 : DINT[20] := ([5] := 6, [6] := 33, [7] := 15, [9] := 15, [10] := 3, [11] := 21, [12] := 45, [13] := 21, [14] := 48, [15] := 6, [16] := 15, [19] := 1);
   LN02_DC_Controlled_Theoretical_Units : BOOL := 1;
   LN02_Door_MNT : DINT;
   LN02_FPY : REAL := 98.0;
   LN02_FrontFrame_MNT : DINT;
   LN02_Ignition_NewSNModel : BOOL[32];
   LN02_Ignition_SNModelMSG : STRING[5] := ([0] := 'WFC150M0JW 3', [1] := 'RC1851273');
   LN02_Last_Message : STRING := 'SHIFT AY ==> 97.69 %';
   LN02_MachineOverAll_MNT : DINT;
   LN02_Main_Messages : DINT[250] := ([4] := 496, [9] := 1, [14] := 10633, [15] := 98, [16] := 18, [17] := 1, [18] := 158, [19] := -11);
   LN02_MainBack_MNT : DINT;
   LN02_MainLine_MSG_Out : MESSAGE;
        MessageParameters(ServiceCode := 16#004d, LocalElement := DC1_to_LN02_Messages[0], ...)
   LN02_Match : DINT;
   LN02_Match_No_Error : DINT;
   LN02_Message_Change : BOOL := 1;
   LN02_Messages_Barcode_SNModel : Barcode_SNModel := (Data[0] := 'WFC150M0JW 3', Data[1] := 'RC1851273');
   LN02_ML_Message : STRING := 'SHIFT AY ==> 97.69 %';
   LN02_MLC_Downtime : BOOL;
   LN02_OT_Shift_Break_In_Minutes : DINT := 60;
   LN02_OvenCavity_MNT : DINT;
   LN02_Schedule : UDT_Current_Status := (Line := 'LN02', Shift := 1, _1st_Shift_Avail := 1, _1st_Shift_Active := 1, _1st_Shift_Scheduled := 1, _2nd_Shift_Scheduled := 1, DayOfWeek := 'Mon', DayOfWeek_Int := 1, Start_Time := '2023-05-08 05:00', End_Time := '2023-05-08 13:30', Scheduled_Units := 1240, Units_Remaining := 782, Units_Produced := 496, Units_Lossed := 40, AY_Percent := 92.79279, Shift_Scheduled := 1, Shift_Active := 1, Theoretical_Units := 597, Running := 1, State := 3, Units_Rejected := 18);
   LN02_Schedule_Cycle_Timer : TIMER := (PRE := 22258, ACC := 6197, EN := 1, TT := 1);
   LN02_Schedule_Max_Break_Duration : DINT := 50;
   LN02_Schedule_Max_Break_Timer : TIMER := (PRE := 3000000, ACC := 649792);
   LN02_Schedule_Tag : STRING := 'SCHED';
   LN02_Schedule_TAKT : DINT := 30000;
   LN02_Schedule_TAKT_REAL : REAL := 22258.064;
   LN02_ScheduleUnits_Produced_from_line : DINT := 51857;
   LN02_SidePanels_MNT : DINT;
   LN02_SNModel_Array : UDT_SN_Model[50] := ([0].LastReadCode := 1, [0].Serial := 'CA0807380', [0].Model := 'WTW4816FW2', [0].DateTime := '2/25/2021 12:28:40.38102', [1].writeIndex := 1, [1].readIndex := 1, [1].LastReadCode := 1, [1].Serial := 'CA0807381', [1].Model := 'WTW4816FW2', [1].DateTime := '2/25/2021 12:28:52.55128', [2].writeIndex := 2, [2].readIndex := 2, [2].LastReadCode := 1, [2].Serial := 'CA0807382', [2].Model := 'WTW4816FW2', [2].DateTime := '2/25/2021 12:29:03.43928', [3].writeIndex := 3, [3].readIndex := 3, [3].LastReadCode := 1, [3].Serial := 'CA0807383', [3].Model := 'WTW4816FW2', [3].DateTime := '2/25/2021 12:29:14.30134', [4].writeIndex := 4, [4].readIndex := 4, [4].LastReadCode := 1, [4].Serial := 'CA0807384', [4].Model := 'WTW4816FW2', [4].DateTime := '2/25/2021 12:29:24.42454', [5].writeIndex := 5, [5].readIndex := 5, [5].LastReadCode := 1, [5].Serial := 'CA0807385', [5].Model := 'WTW4816FW2', [5].DateTime := '2/25/2021 12:29:35.71676', [6].writeIndex := 6, [6].readIndex := 6, [6].LastReadCode := 1, [6].Serial := 'CA0807386', [6].Model := 'WTW4816FW2', [6].DateTime := '2/25/2021 12:29:46.65221', [7].writeIndex := 7, [7].readIndex := 7, [7].LastReadCode := 1, [7].Serial := 'CA0807387', [7].Model := 'WTW4816FW2', [7].DateTime := '2/25/2021 12:29:57.14076', [8].writeIndex := 8, [8].readIndex := 8, [8].LastReadCode := 1, [8].Serial := 'CA0807388', [8].Model := 'WTW4816FW2', [8].DateTime := '2/25/2021 12:30:38.78655', [9].writeIndex := 10, [9].readIndex := 9, [9].LastReadCode := 1, [9].Serial := 'CA0807389', [9].Model := 'WTW4816FW2', [9].DateTime := '2/25/2021 12:30:51.72217', [10].writeIndex := 10, [10].readIndex := 10,
        [10].LastReadCode := 1, [10].Serial := 'CA0807390', [10].Model := 'WTW4816FW2', [10].DateTime := '2/25/2021 12:31:01.80920', [11].writeIndex := 11, [11].readIndex := 11, [11].LastReadCode := 1, [11].Serial := 'CA0807391', [11].Model := 'WTW4816FW2', [11].DateTime := '2/25/2021 12:31:11.91238', [12].writeIndex := 12, [12].readIndex := 12, [12].LastReadCode := 1, [12].Serial := 'CA0807392', [12].Model := 'WTW4816FW2', [12].DateTime := '2/25/2021 12:31:24.82835', [13].writeIndex := 13, [13].readIndex := 13, [13].LastReadCode := 1, [13].Serial := 'CA0807393', [13].Model := 'WTW4816FW2', [13].DateTime := '2/25/2021 12:31:33.33885', [14].writeIndex := 14, [14].readIndex := 14, [14].LastReadCode := 1, [14].Serial := 'CA0807394', [14].Model := 'WTW4816FW2', [14].DateTime := '2/25/2021 12:31:44.26004', [15].writeIndex := 15, [15].readIndex := 15, [15].LastReadCode := 1, [15].Serial := 'CA0807395', [15].Model := 'WTW4816FW2', [15].DateTime := '2/25/2021 12:31:55.17391', [16].writeIndex := 16, [16].readIndex := 16, [16].LastReadCode := 1, [16].Serial := 'CA0807396', [16].Model := 'WTW4816FW2', [16].DateTime := '2/25/2021 12:32:06.90771', [17].writeIndex := 17, [17].readIndex := 17, [17].LastReadCode := 1, [17].Serial := 'CA0807397', [17].Model := 'WTW4816FW2', [17].DateTime := '2/25/2021 12:32:16.96281', [18].writeIndex := 18, [18].readIndex := 18, [18].LastReadCode := 1, [18].Serial := 'CA0807398', [18].Model := 'WTW4816FW2', [18].DateTime := '2/25/2021 12:32:27.92434', [19].writeIndex := 19, [19].readIndex := 19, [19].LastReadCode := 1, [19].Serial := 'CA0807399', [19].Model := 'WTW4816FW2', [19].DateTime := '2/25/2021 12:32:38.40881', [20].writeIndex := 20, [20].readIndex := 20,
        [20].LastReadCode := 1, [20].Serial := 'CA0807400', [20].Model := 'WTW4816FW2', [20].DateTime := '2/25/2021 12:32:49.30917', [21].writeIndex := 21, [21].readIndex := 21, [21].LastReadCode := 1, [21].Serial := 'CA0807401', [21].Model := 'WTW4816FW2', [21].DateTime := '2/25/2021 12:33:00.28133', [22].writeIndex := 22, [22].readIndex := 22, [22].LastReadCode := 1, [22].Serial := 'CA0807402', [22].Model := 'WTW4816FW2', [22].DateTime := '2/25/2021 12:33:35.38591', [23].writeIndex := 23, [23].readIndex := 23, [23].LastReadCode := 1, [23].Serial := 'CA0807403', [23].Model := 'WTW4816FW2', [23].DateTime := '2/25/2021 12:33:45.88840', [24].writeIndex := 24, [24].readIndex := 24, [24].LastReadCode := 1, [24].Serial := 'CA0807404', [24].Model := 'WTW4816FW2', [24].DateTime := '2/25/2021 12:33:56.85644', [25].writeIndex := 25, [25].readIndex := 25, [25].LastReadCode := 1, [25].Serial := 'CA0807405', [25].Model := 'WTW4816FW2', [25].DateTime := '2/25/2021 12:34:07.73473', [26].writeIndex := 26, [26].readIndex := 26, [26].LastReadCode := 1, [26].Serial := 'CA0807406', [26].Model := 'WTW4816FW2', [26].DateTime := '2/25/2021 12:34:18.63707', [27].writeIndex := 27, [27].readIndex := 27, [27].LastReadCode := 1, [27].Serial := 'CA0807407', [27].Model := 'WTW4816FW2', [27].DateTime := '2/25/2021 12:34:29.95757', [28].writeIndex := 28, [28].readIndex := 28, [28].LastReadCode := 1, [28].Serial := 'CA0807408', [28].Model := 'WTW4816FW2', [28].DateTime := '2/25/2021 12:34:41.36491', [29].writeIndex := 29, [29].readIndex := 29, [29].LastReadCode := 1, [29].Serial := 'CA0807409', [29].Model := 'WTW4816FW2', [29].DateTime := '2/25/2021 12:34:52.31039', [30].writeIndex := 30, [30].readIndex := 30,
        [30].LastReadCode := 1, [30].Serial := 'CA0807410', [30].Model := 'WTW4816FW2', [30].DateTime := '2/25/2021 12:35:05.61831', [31].writeIndex := 31, [31].readIndex := 31, [31].LastReadCode := 1, [31].Serial := 'CA0807411', [31].Model := 'WTW4816FW2', [31].DateTime := '2/25/2021 12:35:14.80057', [32].writeIndex := 32, [32].readIndex := 32, [32].LastReadCode := 1, [32].Serial := 'CA0807412', [32].Model := 'WTW4816FW2', [32].DateTime := '2/25/2021 12:35:24.99536', [33].writeIndex := 33, [33].readIndex := 33, [33].LastReadCode := 1, [33].Serial := 'CA0807413', [33].Model := 'WTW4816FW2', [33].DateTime := '2/25/2021 12:35:35.89756', [34].writeIndex := 34, [34].readIndex := 34, [34].LastReadCode := 1, [34].Serial := 'CA0807414', [34].Model := 'WTW4816FW2', [34].DateTime := '2/25/2021 12:35:49.25334', [35].writeIndex := 35, [35].readIndex := 35, [35].LastReadCode := 1, [35].Serial := 'CA0807415', [35].Model := 'WTW4816FW2', [35].DateTime := '2/25/2021 12:35:57.77427', [36].writeIndex := 36, [36].readIndex := 36, [36].LastReadCode := 1, [36].Serial := 'CA0807416', [36].Model := 'WTW4816FW2', [36].DateTime := '2/25/2021 12:36:08.66572', [37].writeIndex := 37, [37].readIndex := 37, [37].LastReadCode := 1, [37].Serial := 'CA0807417', [37].Model := 'WTW4816FW2', [37].DateTime := '2/25/2021 12:36:19.57452', [38].writeIndex := 38, [38].readIndex := 38, [38].LastReadCode := 1, [38].Serial := 'CA0807418', [38].Model := 'WTW4816FW2', [38].DateTime := '2/25/2021 12:36:30.10790', [39].writeIndex := 39, [39].readIndex := 39, [39].LastReadCode := 1, [39].Serial := 'CA0807419', [39].Model := 'WTW4816FW2', [39].DateTime := '2/25/2021 12:36:40.99675', [40].writeIndex := 40, [40].readIndex := 40,
        [40].LastReadCode := 1, [40].Serial := 'CA0807420', [40].Model := 'WTW4816FW2', [40].DateTime := '2/25/2021 12:36:51.92086', [41].writeIndex := 41, [41].readIndex := 41, [41].LastReadCode := 1, [41].Serial := 'CA0807371', [41].Model := 'WTW4816FW2', [41].DateTime := '2/25/2021 12:27:03.39945', [42].writeIndex := 42, [42].readIndex := 42, [42].LastReadCode := 1, [42].Serial := 'CA0807372', [42].Model := 'WTW4816FW2', [42].DateTime := '2/25/2021 12:27:14.31229', [43].writeIndex := 43, [43].readIndex := 43, [43].LastReadCode := 1, [43].Serial := 'CA0807373', [43].Model := 'WTW4816FW2', [43].DateTime := '2/25/2021 12:27:25.22997', [44].writeIndex := 44, [44].readIndex := 44, [44].LastReadCode := 1, [44].Serial := 'CA0807374', [44].Model := 'WTW4816FW2', [44].DateTime := '2/25/2021 12:27:36.12574', [45].writeIndex := 45, [45].readIndex := 45, [45].LastReadCode := 1, [45].Serial := 'CA0807375', [45].Model := 'WTW4816FW2', [45].DateTime := '2/25/2021 12:27:46.64041', [46].writeIndex := 46, [46].readIndex := 46, [46].LastReadCode := 1, [46].Serial := 'CA0807376', [46].Model := 'WTW4816FW2', [46].DateTime := '2/25/2021 12:27:57.56194', [47].writeIndex := 47, [47].readIndex := 47, [47].LastReadCode := 1, [47].Serial := 'CA0807377', [47].Model := 'WTW4816FW2', [47].DateTime := '2/25/2021 12:28:08.50169', [48].writeIndex := 48, [48].readIndex := 48, [48].LastReadCode := 1, [48].Serial := 'CA0807378', [48].Model := 'WTW4816FW2', [48].DateTime := '2/25/2021 12:28:19.39640', [49].writeIndex := 49, [49].readIndex := 49, [49].LastReadCode := 1, [49].Serial := 'CA0807379', [49].Model := 'WTW4816FW2', [49].DateTime := '2/25/2021 12:28:30.29576');
   LN02_SNModel_CurrentRead : UDT_SN_Model := (writeIndex := 38, readIndex := 38, Serial := 'CA0807418', Model := 'WTW4816FW2', DateTime := '2/25/2021 12:36:30.10790');
   LN02_SNModel_STR40 : STRING_40[10] := ([0] := 'CA0807420', [1] := 'WTW4816FW2', [2] := '2/25/2021 12:36:55.546816');
   LN02_Standard_Shift_Break_In_Minutes : DINT := 50;
   LN02_StorageDrawer_MNT : DINT;
   LN02_Test_MNT : DINT;
   LN02_Theoretical_Units_Counter : COUNTER := (PRE := 999999, ACC := 597);
   LN02_Theoretical_Units_Counter_ONS : BOOL;
   LN02_Toggle_CountSource : BOOL := 1;
   LN02_Units_for_repair : DINT := 18;
   LN02_Weekly_Schedule : UDT_Weekly_Schedule := (Monday._1st_Shift_Avail := 1, Monday._1st_Shift_Start := '2023-05-08 05:00', Monday._1st_Shift_End := '2023-05-08 13:30', Monday._2nd_Shift_Avail := 1, Monday._2nd_Shift_Start := '2023-05-08 16:45', Monday._2nd_Shift_End := '2023-05-09 01:15', Monday._3rd_Shift_Start := '2023-05-08 04:50', Monday._3rd_Shift_End := '2023-05-08 04:55', Monday.S1_Scheduled := 1240, Monday.S2_Scheduled := 1240, Tuesday._1st_Shift_Avail := 1, Tuesday._1st_Shift_Start := '2023-05-09 05:00', Tuesday._1st_Shift_End := '2023-05-09 15:30', Tuesday._2nd_Shift_Avail := 1, Tuesday._2nd_Shift_Start := '2023-05-09 16:45', Tuesday._2nd_Shift_End := '2023-05-10 03:15', Tuesday._3rd_Shift_Start := '2023-05-09 04:50', Tuesday._3rd_Shift_End := '2023-05-09 04:55', Tuesday.S1_Scheduled := 1537, Tuesday.S2_Scheduled := 1537, Wednesday._1st_Shift_Avail := 1, Wednesday._1st_Shift_Start := '2023-05-10 05:00', Wednesday._1st_Shift_End := '2023-05-10 15:30', Wednesday._2nd_Shift_Avail := 1, Wednesday._2nd_Shift_Start := '2023-05-10 16:45', Wednesday._2nd_Shift_End := '2023-05-11 03:15', Wednesday._3rd_Shift_Start := '2023-05-10 04:50', Wednesday._3rd_Shift_End := '2023-05-10 04:55', Wednesday.S1_Scheduled := 1537, Wednesday.S2_Scheduled := 1537, Thursday._1st_Shift_Avail := 1, Thursday._1st_Shift_Start := '2023-05-11 05:00', Thursday._1st_Shift_End := '2023-05-11 13:30', Thursday._2nd_Shift_Avail := 1, Thursday._2nd_Shift_Start := '2023-05-11 16:45', Thursday._2nd_Shift_End := '2023-05-12 01:15', Thursday._3rd_Shift_Start := '2023-05-11 04:50', Thursday._3rd_Shift_End := '2023-05-11 04:55', Thursday.S1_Scheduled := 1240, Thursday.S2_Scheduled := 1240, Friday._1st_Shift_Avail := 1, Friday._1st_Shift_Start := '2023-05-12 05:00', Friday._1st_Shift_End := '2023-05-12 13:30', Friday._2nd_Shift_Avail := 1, Friday._2nd_Shift_Start := '2023-05-12 16:45', Friday._2nd_Shift_End := '2023-05-13 01:15', Friday._3rd_Shift_Start := '2023-05-12 04:50', Friday._3rd_Shift_End := '2023-05-12 04:55', Friday.S1_Scheduled := 1240, Friday.S2_Scheduled := 1240, Saturday._1st_Shift_Start := '2023-05-13 05:00', Saturday._1st_Shift_End := '2023-05-13 13:30', Saturday._2nd_Shift_Start := '2023-05-13 16:45', Saturday._2nd_Shift_End := '2023-05-14 01:15', Saturday._3rd_Shift_Start := '2023-05-13 04:50', Saturday._3rd_Shift_End := '2023-05-13 04:55', Sunday._1st_Shift_Start := '2023-05-14 05:00', Sunday._1st_Shift_End := '2023-05-14 13:30', Sunday._2nd_Shift_Start := '2023-05-14 16:45', Sunday._2nd_Shift_End := '2023-05-15 01:15',
        Sunday._3rd_Shift_Start := '2023-05-14 04:50', Sunday._3rd_Shift_End := '2023-05-14 04:55');
   LN02_Wiring_MNT : DINT;
   LN02ECM02 : DINT;
   LN02ECM03 : DINT;
   LN02ECM04 : DINT;
   LN02ECM05 : DINT;
   LN02EDM04 : DINT;
   LN02EDM06 : DINT;
   LN02EDM07 : DINT;
   LN02EDM08 : DINT;
   LN02EEM01 : DINT;
   LN02EEM02 : DINT;
   LN02EEM03 : DINT;
   LN02EES01 : DINT;
   LN02EES02 : DINT;
   LN02EES03 : DINT;
   LN02EES04 : DINT;
   LN02EFS04 : DINT;
   LN02EFS05 : DINT;
   LN02EGM04 : DINT;
   LN02EHM01 : DINT;
   LN02EHM02 : DINT;
   LN02EHM03 : DINT;
   LN02EHM04 : DINT;
   LN02EHM05 : DINT;
   LN02EHM06 : DINT;
   LN02EHM07 : DINT;
   LN02EHM08 : DINT;
   LN02EHM09 : DINT;
   LN02EHM10 : DINT;
   LN02EHM11 : DINT;
   LN02EJM02 : DINT;
   LN02EJM03 : DINT;
   LN02EKM01 : DINT;
   LN02EKM02 : DINT;
   LN02EKM03 : DINT;
   LN02EKM05 : DINT;
   LN02EKM13 : DINT;
   LN02EKM18 : DINT;
   LN02EKM20 : DINT;
   LN02EKM22 : DINT;
   LN02EKM24 : DINT;
   LN02EKM26 : DINT;
   LN02EKM29 : DINT;
   LN02EKM30 : DINT;
   LN02EKM31 : DINT;
   LN02EKM32 : DINT;
   LN02EKM35 : DINT;
   LN02ELM01 : DINT;
   LN02ELM02 : DINT;
   LN02ELM03 : DINT;
   LN02ELM04 : DINT;
   LN02ELM05 : DINT;
   LN02ELS01 : DINT;
   LN02ELS02 : DINT;
   LN02ELS04 : DINT;
   LN02ELS06 : DINT;
   LN02ELS08 : DINT;
   LN02ELS13 : DINT;
   LN02ELS19 : DINT;
   LN02EMM01 : DINT;
   LN02EMM02 : DINT;
   LN02EMM03 : DINT;
   LN02NAS01 : DINT;
   LN02NAS02 : DINT;
   LN02NAS03 : DINT;
   LN02NAS05 : DINT;
   LN02NAS15 : DINT;
   LN02NAS16 : DINT;
   LN02NAS17 : DINT;
   LN02NAS25 : DINT;
   LN02NAS26 : DINT;
   LN02NAS33 : DINT;
   LN02NAS34 : DINT;
   LN02NBS01 : DINT;
   LN02NBS02 : DINT;
   LN02NES01 : DINT;
   LN02NES02 : DINT;
   LN02NES03 : DINT;
   LN02NES04 : DINT;
   LN02NFS01 : DINT;
   LN02NFS02 : DINT;
   LN02NGS06 : DINT;
   LN02NMS01 : DINT;
   LN02SAS01 : DINT;
   LN02SAS02 : DINT;
   LN02SAS03 : DINT;
   LN02SAS11 : DINT;
   LN02SAS13 : DINT;
   LN02SAS29 : DINT;
   LN02SAS35 : DINT;
   LN02SBS01 : DINT;
   LN02SBS02 : DINT;
   LN02SBS03 : DINT;
   LN02SES01 : DINT;
   LN02SES07 : DINT;
   LN02SES08 : DINT;
   LN02SFS01 : DINT;
   LN02SFS02 : DINT;
   LN02SFS03 : DINT;
   LN02SFS04 : DINT;
   LN02SGS01 : DINT;
   LN02SGS07 : DINT;
   LN02SGS08 : DINT;
   LN02SKS05 : DINT;
   LN02SKS06 : DINT;
   LN02SMS09 : DINT;
   LN02WAM01 : DINT;
   LN02WAS35 : DINT;
   LN02WAS42 : DINT;
   LN02WAS44 : DINT;
   LN02WAS45 : DINT;
   LN02WAS46 : DINT;
   LN02WAS48 : DINT;
   LN02WBM01 : DINT;
   LN02WBM02 : DINT;
   LN02WBM03 : DINT;
   LN02WBM04 : DINT;
   LN02WBS06 : DINT;
   LN02WBS12 : DINT;
   LN02WBS13 : DINT;
   LN02WBS26 : DINT;
   LN02WBS32 : DINT;
   LN02WCM01 : DINT;
   LN02WCM02 : DINT;
   LN02WCM03 : DINT;
   LN02WCM04 : DINT;
   LN02WCM05 : DINT;
   LN02WCM06 : DINT;
   LN02WCS06 : DINT;
   LN02WCS07 : DINT;
   LN02WDM01 : DINT;
   LN02WDM02 : DINT;
   LN02WDM03 : DINT;
   LN02WDM04 : DINT;
   LN02WDM05 : DINT;
   LN02WDM06 : DINT;
   LN02WDM10 : DINT;
   LN02WDS03 : DINT;
   LN02WDS06 : DINT;
   LN02WDS11 : DINT;
   LN02WDS14 : DINT;
   LN02WDS15 : DINT;
   LN02WEM01 : DINT;
   LN02WEM09 : DINT;
   LN02WEM09SE : DINT;
   LN02WEM10 : DINT;
   LN02WEM11 : DINT;
   LN02WEM12 : DINT;
   LN02WEM12SA : DINT;
   LN02WEM12SB : DINT;
   LN02WEM12SB1 : DINT;
   LN02WEM12SC : DINT;
   LN02WEM15 : DINT;
   LN02WEM15SA : DINT;
   LN02WEM15SB : DINT;
   LN02WEM22 : DINT;
   LN02WEM31 : DINT;
   LN02WEM31SF : DINT;
   LN02WFM01 : DINT;
   LN02WFS01 : DINT;
   LN02WFS02 : DINT;
   LN02WFS12 : DINT;
   LN02WFS13 : DINT;
   LN02WFS17 : DINT;
   LN02WFS18 : DINT;
   LN02WGM01 : DINT;
   LN02WGM02 : DINT;
   LN02WGM03 : DINT;
   LN02WGM04 : DINT;
   LN02WGM05 : DINT;
   LN02WGS01 : DINT;
   LN02WGS02 : DINT;
   LN02WGS03 : DINT;
   LN02WGS04 : DINT;
   LN02WHM08 : DINT;
   LN02WHM09 : DINT;
   LN02WHM10 : DINT;
   LN02WHS01 : DINT;
   LN02WJM11 : DINT;
   LN02WJM16 : DINT;
   LN02WJM18 : DINT;
   LN02WJM19 : DINT;
   LN02WJM21 : DINT;
   LN02WJM28 : DINT;
   LN02WJM31 : DINT;
   LN02WJM32 : DINT;
   LN02WJM33 : DINT;
   LN02WJM42 : DINT;
   LN02WJM46 : DINT;
   LN02WJM60 : DINT;
   LN02WJM60BL1 : DINT;
   LN02WJM60BL2 : DINT;
   LN02WJM60BL3 : DINT;
   LN02WJM60BL4 : DINT;
   LN02WJS01 : DINT;
   LN02WJS02 : DINT;
   LN02WJS03 : DINT;
   LN02WKM01 : DINT;
   LN02WKS01 : DINT;
   LN02WKS02 : DINT;
   LN02WKS03 : DINT;
   LN02WKS04 : DINT;
   LN02WKS05 : DINT;
   LN02WLM06 : DINT;
   LN02WLM07 : DINT;
   LN02WLS04 : DINT;
   LN02WMM02 : DINT;
   LN02WMM03 : DINT;
   LN02XAS01 : DINT;
   LN02XAS02 : DINT;
   LN02XAS03 : DINT;
   LN02XAS04 : DINT;
   LN02XAS05 : DINT;
   LN02XAS06 : DINT;
   LN02XBS01 : DINT;
   LN02XBS02 : DINT;
   LN02XBS03 : DINT;
   LN02XCS01 : DINT;
   LN02XCS02 : DINT;
   LN02XCS03 : DINT;
   LN02XDM01 : DINT;
   LN02XDM02 : DINT;
   LN02XDM03 : DINT;
   LN02XDS01 : DINT;
   LN02XDS02 : DINT;
   LN02XDS03 : DINT;
   LN02XEM01 : DINT;
   LN02XEM02 : DINT;
   LN02XEM03 : DINT;
   LN02XES01 : DINT;
   LN02XES02 : DINT;
   LN02XES03 : DINT;
   LN02XFS01 : DINT;
   LN02XFS02 : DINT;
   LN02XFS03 : DINT;
   LN02XGS01 : DINT;
   LN02XGS02 : DINT;
   LN02XGS03 : DINT;
   LN02XHS01 : DINT;
   LN02XHS02 : DINT;
   LN02XHS03 : DINT;
   LN02XIM01 : DINT;
   LN02XIM02 : DINT;
   LN02XIM03 : DINT;
   LN02XJM01 : DINT;
   LN02XJM02 : DINT;
   LN02XJM03 : DINT;
   LN02XKM01 : DINT;
   LN02XKM02 : DINT;
   LN02XKM03 : DINT;
   LN02XLS01 : DINT;
   LN02XLS02 : DINT;
   LN02XLS03 : DINT;
   LN02XMS01 : DINT;
   LN02XMS02 : DINT;
   LN02XMS03 : DINT;
   LN02ZMN01 : DINT;
   LN02ZMN02 : DINT;
   LN02ZMN03 : DINT;
   LN02ZMN04 : DINT;
   LN02ZMS01 : DINT;
   LN02ZMS02 : DINT;
   LN02ZMS03 : DINT;
   LN02ZMS04 : DINT;
   LN03_1st_Station_Break_Code : DINT := 16;
   LN03_Additional_Break_Limit_Mins : DINT := 570;
   LN03_assist1 : DINT;
   LN03_assist2 : DINT;
   LN03_assist3 : DINT;
   LN03_assist4 : DINT;
   LN03_Assist_CT : DINT;
   LN03_Assist_Record : STRING := '02EDM-35';
   LN03_Assist_Tag : STRING := 'ASSIST';
   LN03_Assist_Tags : STRING[5];
   LN03_AY : REAL := 0.8739003;
   LN03_Boxing_MNT : DINT;
   LN03_Console_MNT : DINT;
   LN03_Cooktop_MNT : DINT;
   LN03_Current_Shift_Duration_Mins : DINT := 510;   // CURRENT SHIFT TOTAL MINUTES SCHEDULED
   LN03_Current_Shift_Duration_wBreaks_Mins : DINT := 460;
   LN03_DataFromDC1 : DINT[20] := ([5] := 20, [6] := 3, [7] := 20, [8] := 3, [9] := 20, [10] := 3, [11] := 20, [12] := 3, [13] := 20, [14] := 3, [15] := 20, [16] := 3);
   LN03_DataFromDC3 : DINT[20] := ([5] := 6, [6] := 33, [7] := 15, [9] := 15, [10] := 3, [11] := 21, [12] := 45, [13] := 21, [14] := 48, [15] := 6, [16] := 15);
   LN03_DC_Controlled_Theoretical_Units : BOOL := 1;
   LN03_Door_MNT : DINT;
   LN03_FPY : REAL := 97.0;
   LN03_FrontFrame_MNT : DINT;
   LN03_Ignition_NewSNModel : BOOL[32];
   LN03_Ignition_SNModelMSG : STRING[5];
   LN03_Last_Message : STRING := 'SHIFT AY ==> 97.69 %';
   LN03_LeakTest_MNT : DINT;
   LN03_MachineOverAll_MNT : DINT;
   LN03_Main_Messages : DINT[250] := ([4] := 275, [9] := 1, [15] := 97, [16] := 20, [17] := 1, [18] := 699, [19] := 52);
        [9].1   // BREAK SCHEDULED LINE NOT IN PRODUCTION
        [9].0   // LINE CURRENTLY IN PRODUCTION
   LN03_MainBack_MNT : DINT;
   LN03_MainLine_MSG_Out : MESSAGE;   // Data Messages From Data Concentrator 1 To Assembly Line 3
        MessageParameters(ServiceCode := 16#004d, LocalElement := DC1_to_LN03_Messages[0], ...)
   LN03_Match : DINT;
   LN03_Match_No_Error : DINT;
   LN03_Message_Change : BOOL := 1;
   LN03_Messages_Barcode_SNModel : Barcode_SNModel;
   LN03_ML_Message : STRING := 'SHIFT AY ==> 97.69 %';
   LN03_MLC_Downtime : BOOL;
   LN03_OT_Shift_Break_In_Minutes : DINT := 60;
   LN03_OvenCavity_MNT : DINT;
   LN03_Schedule : UDT_Current_Status := (Line := 'LN03', Shift := 1, _1st_Shift_Avail := 1, _1st_Shift_Active := 1, _1st_Shift_Scheduled := 1, _2nd_Shift_Scheduled := 1, DayOfWeek := 'Mon', DayOfWeek_Int := 1, Start_Time := '2023-05-08 05:00', End_Time := '2023-05-08 13:30', Scheduled_Units := 700, Units_Remaining := 462, Units_Produced := 275, Units_Lossed := 43, AY_Percent := 87.39003, Shift_Scheduled := 1, Shift_Active := 1, Theoretical_Units := 337, Running := 1, State := 3, Units_Rejected := 20);
        .Shift   // CURRENT SHIFT SCHEDULED
        .Shift_Active   // CURRENT SHIFT PRODUCTION SCHEDULED
        .Theoretical_Units   // CURRENT NUMBER OF UNITS THAT SHOULD BE BUILT
   LN03_Schedule_Cycle_Timer : TIMER := (PRE := 39429, ACC := 8214, EN := 1, TT := 1);   // UNIT CYCLE ( TAKT TIME ) TIMER
   LN03_Schedule_Max_Break_Duration : DINT := 50;
   LN03_Schedule_Max_Break_Timer : TIMER := (PRE := 3000000, ACC := 648907);
   LN03_Schedule_Tag : STRING := 'SCHED';
   LN03_Schedule_TAKT : REAL := 39428.57;
   LN03_ScheduleUnits_Produced_from_line : DINT := 16273;
   LN03_SidePanels_MNT : DINT;
   LN03_SNModel_Array : UDT_SN_Model[50] := ([0].LastReadCode := 1, [0].Serial := 'CA0807380', [0].Model := 'WTW4816FW2', [0].DateTime := '2/25/2021 12:28:40.38102', [1].writeIndex := 1, [1].readIndex := 1, [1].LastReadCode := 1, [1].Serial := 'CA0807381', [1].Model := 'WTW4816FW2', [1].DateTime := '2/25/2021 12:28:52.55128', [2].writeIndex := 2, [2].readIndex := 2, [2].LastReadCode := 1, [2].Serial := 'CA0807382', [2].Model := 'WTW4816FW2', [2].DateTime := '2/25/2021 12:29:03.43928', [3].writeIndex := 3, [3].readIndex := 3, [3].LastReadCode := 1, [3].Serial := 'CA0807383', [3].Model := 'WTW4816FW2', [3].DateTime := '2/25/2021 12:29:14.30134', [4].writeIndex := 4, [4].readIndex := 4, [4].LastReadCode := 1, [4].Serial := 'CA0807384', [4].Model := 'WTW4816FW2', [4].DateTime := '2/25/2021 12:29:24.42454', [5].writeIndex := 5, [5].readIndex := 5, [5].LastReadCode := 1, [5].Serial := 'CA0807385', [5].Model := 'WTW4816FW2', [5].DateTime := '2/25/2021 12:29:35.71676', [6].writeIndex := 6, [6].readIndex := 6, [6].LastReadCode := 1, [6].Serial := 'CA0807386', [6].Model := 'WTW4816FW2', [6].DateTime := '2/25/2021 12:29:46.65221', [7].writeIndex := 7, [7].readIndex := 7, [7].LastReadCode := 1, [7].Serial := 'CA0807387', [7].Model := 'WTW4816FW2', [7].DateTime := '2/25/2021 12:29:57.14076', [8].writeIndex := 8, [8].readIndex := 8, [8].LastReadCode := 1, [8].Serial := 'CA0807388', [8].Model := 'WTW4816FW2', [8].DateTime := '2/25/2021 12:30:38.78655', [9].writeIndex := 10, [9].readIndex := 9, [9].LastReadCode := 1, [9].Serial := 'CA0807389', [9].Model := 'WTW4816FW2', [9].DateTime := '2/25/2021 12:30:51.72217', [10].writeIndex := 10, [10].readIndex := 10,
        [10].LastReadCode := 1, [10].Serial := 'CA0807390', [10].Model := 'WTW4816FW2', [10].DateTime := '2/25/2021 12:31:01.80920', [11].writeIndex := 11, [11].readIndex := 11, [11].LastReadCode := 1, [11].Serial := 'CA0807391', [11].Model := 'WTW4816FW2', [11].DateTime := '2/25/2021 12:31:11.91238', [12].writeIndex := 12, [12].readIndex := 12, [12].LastReadCode := 1, [12].Serial := 'CA0807392', [12].Model := 'WTW4816FW2', [12].DateTime := '2/25/2021 12:31:24.82835', [13].writeIndex := 13, [13].readIndex := 13, [13].LastReadCode := 1, [13].Serial := 'CA0807393', [13].Model := 'WTW4816FW2', [13].DateTime := '2/25/2021 12:31:33.33885', [14].writeIndex := 14, [14].readIndex := 14, [14].LastReadCode := 1, [14].Serial := 'CA0807394', [14].Model := 'WTW4816FW2', [14].DateTime := '2/25/2021 12:31:44.26004', [15].writeIndex := 15, [15].readIndex := 15, [15].LastReadCode := 1, [15].Serial := 'CA0807395', [15].Model := 'WTW4816FW2', [15].DateTime := '2/25/2021 12:31:55.17391', [16].writeIndex := 16, [16].readIndex := 16, [16].LastReadCode := 1, [16].Serial := 'CA0807396', [16].Model := 'WTW4816FW2', [16].DateTime := '2/25/2021 12:32:06.90771', [17].writeIndex := 17, [17].readIndex := 17, [17].LastReadCode := 1, [17].Serial := 'CA0807397', [17].Model := 'WTW4816FW2', [17].DateTime := '2/25/2021 12:32:16.96281', [18].writeIndex := 18, [18].readIndex := 18, [18].LastReadCode := 1, [18].Serial := 'CA0807398', [18].Model := 'WTW4816FW2', [18].DateTime := '2/25/2021 12:32:27.92434', [19].writeIndex := 19, [19].readIndex := 19, [19].LastReadCode := 1, [19].Serial := 'CA0807399', [19].Model := 'WTW4816FW2', [19].DateTime := '2/25/2021 12:32:38.40881', [20].writeIndex := 20, [20].readIndex := 20,
        [20].LastReadCode := 1, [20].Serial := 'CA0807400', [20].Model := 'WTW4816FW2', [20].DateTime := '2/25/2021 12:32:49.30917', [21].writeIndex := 21, [21].readIndex := 21, [21].LastReadCode := 1, [21].Serial := 'CA0807401', [21].Model := 'WTW4816FW2', [21].DateTime := '2/25/2021 12:33:00.28133', [22].writeIndex := 22, [22].readIndex := 22, [22].LastReadCode := 1, [22].Serial := 'CA0807402', [22].Model := 'WTW4816FW2', [22].DateTime := '2/25/2021 12:33:35.38591', [23].writeIndex := 23, [23].readIndex := 23, [23].LastReadCode := 1, [23].Serial := 'CA0807403', [23].Model := 'WTW4816FW2', [23].DateTime := '2/25/2021 12:33:45.88840', [24].writeIndex := 24, [24].readIndex := 24, [24].LastReadCode := 1, [24].Serial := 'CA0807404', [24].Model := 'WTW4816FW2', [24].DateTime := '2/25/2021 12:33:56.85644', [25].writeIndex := 25, [25].readIndex := 25, [25].LastReadCode := 1, [25].Serial := 'CA0807405', [25].Model := 'WTW4816FW2', [25].DateTime := '2/25/2021 12:34:07.73473', [26].writeIndex := 26, [26].readIndex := 26, [26].LastReadCode := 1, [26].Serial := 'CA0807406', [26].Model := 'WTW4816FW2', [26].DateTime := '2/25/2021 12:34:18.63707', [27].writeIndex := 27, [27].readIndex := 27, [27].LastReadCode := 1, [27].Serial := 'CA0807407', [27].Model := 'WTW4816FW2', [27].DateTime := '2/25/2021 12:34:29.95757', [28].writeIndex := 28, [28].readIndex := 28, [28].LastReadCode := 1, [28].Serial := 'CA0807408', [28].Model := 'WTW4816FW2', [28].DateTime := '2/25/2021 12:34:41.36491', [29].writeIndex := 29, [29].readIndex := 29, [29].LastReadCode := 1, [29].Serial := 'CA0807409', [29].Model := 'WTW4816FW2', [29].DateTime := '2/25/2021 12:34:52.31039', [30].writeIndex := 30, [30].readIndex := 30,
        [30].LastReadCode := 1, [30].Serial := 'CA0807410', [30].Model := 'WTW4816FW2', [30].DateTime := '2/25/2021 12:35:05.61831', [31].writeIndex := 31, [31].readIndex := 31, [31].LastReadCode := 1, [31].Serial := 'CA0807411', [31].Model := 'WTW4816FW2', [31].DateTime := '2/25/2021 12:35:14.80057', [32].writeIndex := 32, [32].readIndex := 32, [32].LastReadCode := 1, [32].Serial := 'CA0807412', [32].Model := 'WTW4816FW2', [32].DateTime := '2/25/2021 12:35:24.99536', [33].writeIndex := 33, [33].readIndex := 33, [33].LastReadCode := 1, [33].Serial := 'CA0807413', [33].Model := 'WTW4816FW2', [33].DateTime := '2/25/2021 12:35:35.89756', [34].writeIndex := 34, [34].readIndex := 34, [34].LastReadCode := 1, [34].Serial := 'CA0807414', [34].Model := 'WTW4816FW2', [34].DateTime := '2/25/2021 12:35:49.25334', [35].writeIndex := 35, [35].readIndex := 35, [35].LastReadCode := 1, [35].Serial := 'CA0807415', [35].Model := 'WTW4816FW2', [35].DateTime := '2/25/2021 12:35:57.77427', [36].writeIndex := 36, [36].readIndex := 36, [36].LastReadCode := 1, [36].Serial := 'CA0807416', [36].Model := 'WTW4816FW2', [36].DateTime := '2/25/2021 12:36:08.66572', [37].writeIndex := 37, [37].readIndex := 37, [37].LastReadCode := 1, [37].Serial := 'CA0807417', [37].Model := 'WTW4816FW2', [37].DateTime := '2/25/2021 12:36:19.57452', [38].writeIndex := 38, [38].readIndex := 38, [38].LastReadCode := 1, [38].Serial := 'CA0807418', [38].Model := 'WTW4816FW2', [38].DateTime := '2/25/2021 12:36:30.10790', [39].writeIndex := 39, [39].readIndex := 39, [39].LastReadCode := 1, [39].Serial := 'CA0807419', [39].Model := 'WTW4816FW2', [39].DateTime := '2/25/2021 12:36:40.99675', [40].writeIndex := 40, [40].readIndex := 40,
        [40].LastReadCode := 1, [40].Serial := 'CA0807420', [40].Model := 'WTW4816FW2', [40].DateTime := '2/25/2021 12:36:51.92086', [41].writeIndex := 41, [41].readIndex := 41, [41].LastReadCode := 1, [41].Serial := 'CA0807371', [41].Model := 'WTW4816FW2', [41].DateTime := '2/25/2021 12:27:03.39945', [42].writeIndex := 42, [42].readIndex := 42, [42].LastReadCode := 1, [42].Serial := 'CA0807372', [42].Model := 'WTW4816FW2', [42].DateTime := '2/25/2021 12:27:14.31229', [43].writeIndex := 43, [43].readIndex := 43, [43].LastReadCode := 1, [43].Serial := 'CA0807373', [43].Model := 'WTW4816FW2', [43].DateTime := '2/25/2021 12:27:25.22997', [44].writeIndex := 44, [44].readIndex := 44, [44].LastReadCode := 1, [44].Serial := 'CA0807374', [44].Model := 'WTW4816FW2', [44].DateTime := '2/25/2021 12:27:36.12574', [45].writeIndex := 45, [45].readIndex := 45, [45].LastReadCode := 1, [45].Serial := 'CA0807375', [45].Model := 'WTW4816FW2', [45].DateTime := '2/25/2021 12:27:46.64041', [46].writeIndex := 46, [46].readIndex := 46, [46].LastReadCode := 1, [46].Serial := 'CA0807376', [46].Model := 'WTW4816FW2', [46].DateTime := '2/25/2021 12:27:57.56194', [47].writeIndex := 47, [47].readIndex := 47, [47].LastReadCode := 1, [47].Serial := 'CA0807377', [47].Model := 'WTW4816FW2', [47].DateTime := '2/25/2021 12:28:08.50169', [48].writeIndex := 48, [48].readIndex := 48, [48].LastReadCode := 1, [48].Serial := 'CA0807378', [48].Model := 'WTW4816FW2', [48].DateTime := '2/25/2021 12:28:19.39640', [49].writeIndex := 49, [49].readIndex := 49, [49].LastReadCode := 1, [49].Serial := 'CA0807379', [49].Model := 'WTW4816FW2', [49].DateTime := '2/25/2021 12:28:30.29576');
   LN03_SNModel_CurrentRead : UDT_SN_Model := (writeIndex := 38, readIndex := 38, Serial := 'CA0807418', Model := 'WTW4816FW2', DateTime := '2/25/2021 12:36:30.10790');
   LN03_SNModel_STR40 : STRING_40[10] := ([0] := 'CA0807420', [1] := 'WTW4816FW2', [2] := '2/25/2021 12:36:55.546816');
   LN03_Standard_Shift_Break_In_Minutes : DINT := 50;
   LN03_StorageDrawer_MNT : DINT;
   LN03_Test_MNT : DINT;
   LN03_Theoretical_Units_Counter : COUNTER := (PRE := 999999, ACC := 337);   // CURRENT NUMBER OF UNITS THAT SHOULD BE BUILT
   LN03_Theoretical_Units_Counter_ONS : BOOL;
   LN03_Toggle_CountSource : BOOL := 1;
   LN03_Units_for_repair : DINT := 97;
   LN03_Weekly_Schedule : UDT_Weekly_Schedule := (Monday._1st_Shift_Avail := 1, Monday._1st_Shift_Start := '2023-05-08 05:00', Monday._1st_Shift_End := '2023-05-08 13:30', Monday._2nd_Shift_Avail := 1, Monday._2nd_Shift_Start := '2023-05-08 16:45', Monday._2nd_Shift_End := '2023-05-09 01:15', Monday._3rd_Shift_Start := '2023-05-08 04:50', Monday._3rd_Shift_End := '2023-05-08 04:55', Monday.S1_Scheduled := 700, Monday.S2_Scheduled := 700, Tuesday._1st_Shift_Avail := 1, Tuesday._1st_Shift_Start := '2023-05-09 05:00', Tuesday._1st_Shift_End := '2023-05-09 15:30', Tuesday._2nd_Shift_Avail := 1, Tuesday._2nd_Shift_Start := '2023-05-09 16:45', Tuesday._2nd_Shift_End := '2023-05-10 01:15', Tuesday._3rd_Shift_Start := '2023-05-09 04:50', Tuesday._3rd_Shift_End := '2023-05-09 04:55', Tuesday.S1_Scheduled := 868, Tuesday.S2_Scheduled := 700, Wednesday._1st_Shift_Avail := 1, Wednesday._1st_Shift_Start := '2023-05-10 05:00', Wednesday._1st_Shift_End := '2023-05-10 15:30', Wednesday._2nd_Shift_Avail := 1, Wednesday._2nd_Shift_Start := '2023-05-10 16:45', Wednesday._2nd_Shift_End := '2023-05-11 01:15', Wednesday._3rd_Shift_Start := '2023-05-10 04:50', Wednesday._3rd_Shift_End := '2023-05-10 04:55', Wednesday.S1_Scheduled := 868, Wednesday.S2_Scheduled := 700, Thursday._1st_Shift_Avail := 1, Thursday._1st_Shift_Start := '2023-05-11 05:00', Thursday._1st_Shift_End := '2023-05-11 13:30', Thursday._2nd_Shift_Avail := 1, Thursday._2nd_Shift_Start := '2023-05-11 16:45', Thursday._2nd_Shift_End := '2023-05-12 01:15', Thursday._3rd_Shift_Start := '2023-05-11 04:50', Thursday._3rd_Shift_End := '2023-05-11 04:55', Thursday.S1_Scheduled := 700, Thursday.S2_Scheduled := 700, Friday._1st_Shift_Avail := 1, Friday._1st_Shift_Start := '2023-05-12 05:00', Friday._1st_Shift_End := '2023-05-12 13:30', Friday._2nd_Shift_Avail := 1, Friday._2nd_Shift_Start := '2023-05-12 16:45', Friday._2nd_Shift_End := '2023-05-13 01:15', Friday._3rd_Shift_Start := '2023-05-12 04:50', Friday._3rd_Shift_End := '2023-05-12 04:55', Friday.S1_Scheduled := 700, Friday.S2_Scheduled := 700, Saturday._1st_Shift_Start := '2023-05-13 05:00', Saturday._1st_Shift_End := '2023-05-13 13:30', Saturday._2nd_Shift_Start := '2023-05-13 16:45', Saturday._2nd_Shift_End := '2023-05-13 23:55', Saturday._3rd_Shift_Start := '2023-05-13 04:50', Saturday._3rd_Shift_End := '2023-05-13 04:55', Sunday._1st_Shift_Start := '2023-05-14 05:00', Sunday._1st_Shift_End := '2023-05-14 13:30', Sunday._2nd_Shift_Start := '2023-05-14 16:45', Sunday._2nd_Shift_End := '2023-05-14 23:55',
        Sunday._3rd_Shift_Start := '2023-05-14 04:50', Sunday._3rd_Shift_End := '2023-05-14 04:55');
   LN03_Wiring_MNT : DINT;
   LN03ECM01 : DINT;
   LN03ECM02 : DINT;
   LN03ECM03 : DINT;
   LN03ECM04 : DINT;
   LN03ECM05 : DINT;
   LN03ECM06 : DINT;
   LN03EDM04 : DINT;
   LN03EDM06 : DINT;
   LN03EDM07 : DINT;
   LN03EDM08 : DINT;
   LN03EEM01 : DINT;
   LN03EEM02 : DINT;
   LN03EEM03 : DINT;
   LN03EES01 : DINT;
   LN03EES02 : DINT;
   LN03EES03 : DINT;
   LN03EES04 : DINT;
   LN03EFS04 : DINT;
   LN03EFS05 : DINT;
   LN03EGM01 : DINT;
   LN03EGM02 : DINT;
   LN03EGM04 : DINT;
   LN03EHM01 : DINT;
   LN03EHM02 : DINT;
   LN03EHM03 : DINT;
   LN03EHM04 : DINT;
   LN03EHM05 : DINT;
   LN03EHM06 : DINT;
   LN03EHM07 : DINT;
   LN03EHM08 : DINT;
   LN03EJM02 : DINT;
   LN03EJM03 : DINT;
   LN03EKM01 : DINT;
   LN03EKM02 : DINT;
   LN03EKM03 : DINT;
   LN03ELM01 : DINT;
   LN03ELM02 : DINT;
   LN03ELM03 : DINT;
   LN03ELM04 : DINT;
   LN03ELM05 : DINT;
   LN03EMM01 : DINT;
   LN03EMM02 : DINT;
   LN03EMM03 : DINT;
   LN03NAS01 : DINT;
   LN03NAS02 : DINT;
   LN03NAS03 : DINT;
   LN03NAS04 : DINT;
   LN03NBS02 : DINT;
   LN03NBS03 : DINT;
   LN03NCS01 : DINT;
   LN03NCS02 : DINT;
   LN03NCS03 : DINT;
   LN03NCS04 : DINT;
   LN03NCS05 : DINT;
   LN03NFS01 : DINT;
   LN03NFS03 : DINT;
   LN03SAS03 : DINT;
   LN03SBS01 : DINT;
   LN03SBS02 : DINT;
   LN03SBS03 : DINT;
   LN03SCS03 : DINT;
   LN03SES01 : DINT;
   LN03SFS01 : DINT;
   LN03SFS02 : DINT;
   LN03SFS03 : DINT;
   LN03SFS04 : DINT;
   LN03SKS05 : DINT;
   LN03WAM01 : DINT;
   LN03WBM01 : DINT;
   LN03WBM02 : DINT;
   LN03WBM03 : DINT;
   LN03WBM04 : DINT;
   LN03WCM01 : DINT;
   LN03WCM02 : DINT;
   LN03WCM03 : DINT;
   LN03WCM04 : DINT;
   LN03WCM05 : DINT;
   LN03WCM06 : DINT;
   LN03WDM01 : DINT;
   LN03WDM02 : DINT;
   LN03WDM03 : DINT;
   LN03WDM04 : DINT;
   LN03WDM05 : DINT;
   LN03WEM01 : DINT;
   LN03WEM02 : DINT;
   LN03WFM01 : DINT;
   LN03WFM02 : DINT;
   LN03WFM03 : DINT;
   LN03WFM04 : DINT;
   LN03WFM05 : DINT;
   LN03WFM06 : DINT;
   LN03WFS01 : DINT;
   LN03WFS02 : DINT;
   LN03WGM01 : DINT;
   LN03WGM02 : DINT;
   LN03WGM03 : DINT;
   LN03WGM04 : DINT;
   LN03WGM05 : DINT;
   LN03WHM02 : DINT;
   LN03WHM08 : DINT;
   LN03WHM09 : DINT;
   LN03WJS01 : DINT;
   LN03WJS02 : DINT;
   LN03WJS03 : DINT;
   LN03WJS04 : DINT;
   LN03WJS05 : DINT;
   LN03WKS01 : DINT;
   LN03WKS02 : DINT;
   LN03WKS03 : DINT;
   LN03WKS04 : DINT;
   LN03WKS05 : DINT;
   LN03WLM02 : DINT;
   LN03WLM04 : DINT;
   LN03WLM06 : DINT;
   LN03WLM07 : DINT;
   LN03WMM02 : DINT;
   LN03ZMN01 : DINT;
   LN03ZMN02 : DINT;
   LN03ZMN03 : DINT;
   LN03ZMN04 : DINT;
   LN03ZMS01 : DINT;
   LN03ZMS02 : DINT;
   LN03ZMS03 : DINT;
   LN03ZMS04 : DINT;
   LN04_1st_Station_Break_Code : DINT := 16;
   LN04_Additional_Break_Limit_Mins : DINT := 570;
   LN04_assist1 : DINT;
   LN04_assist2 : DINT;
   LN04_assist3 : DINT;
   LN04_assist4 : DINT;
   LN04_Assist_CT : DINT;
   LN04_Assist_Record : STRING := '02EDM-35';
   LN04_Assist_Tag : STRING := 'ASSIST';
   LN04_Assist_Tags : STRING[5];
   LN04_BakeDrawer_MNT : DINT;
   LN04_Boxing_MNT : DINT;
   LN04_Console_MNT : DINT;
   LN04_Cooktop_MNT : DINT;
   LN04_Current_Shift_Duration_Mins : DINT := 510;
   LN04_Current_Shift_Duration_wBreaks_Mins : DINT := 460;
   LN04_Data_MSG_Out : MESSAGE;
        MessageParameters(ServiceCode := 16#004d, LocalElement := DC01_to_LN04_Data[0], ...)
   LN04_DataFromDC1 : DINT[20] := ([2] := 1, [5] := 20, [6] := 3, [7] := 20, [8] := 3, [9] := 20, [10] := 3, [11] := 20, [12] := 3, [13] := 20, [14] := 3, [15] := 20, [16] := 3);
   LN04_DataFromDC3 : DINT[20] := ([5] := 6, [6] := 33, [7] := 15, [9] := 15, [10] := 3, [11] := 21, [12] := 45, [13] := 21, [14] := 48, [15] := 6, [16] := 15);
   LN04_DC_Controlled_Theoretical_Units : BOOL := 1;
   LN04_Door_MNT : DINT;
   LN04_EStop_Funct_Test : DINT;
   LN04_EStop_Main_Panel : DINT;
   LN04_EStop_Main_Safety_Relay : DINT;
   LN04_EStop_MCC_Cabinet : DINT;
   LN04_FPY : REAL := 100.0;
   LN04_FrontFrame_MNT : DINT;
   LN04_FunctionalTest_MNT : DINT;
   LN04_Ignition_NewSNModel : BOOL[32];
   LN04_Ignition_SNModelMSG : STRING[5];
   LN04_Last_Message : STRING := 'SHIFT AY ==> 97.69 %';
   LN04_MachineOverAll_MNT : DINT;
   LN04_Main_Messages : DINT[250] := ([4] := 185, [9] := 1, [14] := 101, [15] := 100, [16] := 22, [17] := 1, [18] := 398, [19] := 392);
   LN04_MainBack_MNT : DINT;
   LN04_MainLine_MSG_Out : MESSAGE;
        MessageParameters(ServiceCode := 16#004d, LocalElement := DC1_to_LN04_Messages[0], ...)
   LN04_Match : DINT;
   LN04_Match_No_Error : DINT;
   LN04_Message_Change : BOOL := 1;
   LN04_Messages_Barcode_SNModel : Barcode_SNModel;
   LN04_ML_Message : STRING := 'SHIFT AY ==> 97.69 %';
   LN04_MLC_Downtime : BOOL;
   LN04_OT_Shift_Break_In_Minutes : DINT := 60;
   LN04_OvenCavity_MNT : DINT;
   LN04_Pull_Cord_EStop_9111 : DINT;
   LN04_Pull_Cord_EStop_9112 : DINT;
   LN04_Pull_Cord_EStop_9200 : DINT;
   LN04_Pull_Cord_EStop_9201 : DINT;
   LN04_RackAndLiterature_MNT : DINT;
   LN04_Schedule : UDT_Current_Status := (Line := 'LN04', Shift := 1, _1st_Shift_Avail := 1, _1st_Shift_Active := 1, _1st_Shift_Scheduled := 1, DayOfWeek := 'Mon', DayOfWeek_Int := 1, Start_Time := '2023-05-08 05:00', End_Time := '2023-05-08 13:30', Scheduled_Units := 425, Units_Remaining := 281, Units_Produced := 185, Units_Lossed := 24, AY_Percent := 88.679245, Shift_Scheduled := 1, Shift_Active := 1, Theoretical_Units := 204, Running := 1, State := 3, Units_Rejected := 22);
   LN04_Schedule_Cycle_Timer : TIMER := (PRE := 64941, ACC := 48244, EN := 1, TT := 1);
   LN04_Schedule_Max_Break_Duration : DINT := 50;
   LN04_Schedule_Max_Break_Timer : TIMER := (PRE := 3000000, ACC := 648942);
   LN04_Schedule_Tag : STRING := 'SCHED';
   LN04_Schedule_TAKT : REAL := 64941.176;
   LN04_ScheduleUnits_Produced_from_line : DINT := 7613;
   LN04_SidePanel_MNT : DINT;
   LN04_SNModel_Array : UDT_SN_Model[50] := ([0].LastReadCode := 1, [0].Serial := 'CA0807380', [0].Model := 'WTW4816FW2', [0].DateTime := '2/25/2021 12:28:40.38102', [1].writeIndex := 1, [1].readIndex := 1, [1].LastReadCode := 1, [1].Serial := 'CA0807381', [1].Model := 'WTW4816FW2', [1].DateTime := '2/25/2021 12:28:52.55128', [2].writeIndex := 2, [2].readIndex := 2, [2].LastReadCode := 1, [2].Serial := 'CA0807382', [2].Model := 'WTW4816FW2', [2].DateTime := '2/25/2021 12:29:03.43928', [3].writeIndex := 3, [3].readIndex := 3, [3].LastReadCode := 1, [3].Serial := 'CA0807383', [3].Model := 'WTW4816FW2', [3].DateTime := '2/25/2021 12:29:14.30134', [4].writeIndex := 4, [4].readIndex := 4, [4].LastReadCode := 1, [4].Serial := 'CA0807384', [4].Model := 'WTW4816FW2', [4].DateTime := '2/25/2021 12:29:24.42454', [5].writeIndex := 5, [5].readIndex := 5, [5].LastReadCode := 1, [5].Serial := 'CA0807385', [5].Model := 'WTW4816FW2', [5].DateTime := '2/25/2021 12:29:35.71676', [6].writeIndex := 6, [6].readIndex := 6, [6].LastReadCode := 1, [6].Serial := 'CA0807386', [6].Model := 'WTW4816FW2', [6].DateTime := '2/25/2021 12:29:46.65221', [7].writeIndex := 7, [7].readIndex := 7, [7].LastReadCode := 1, [7].Serial := 'CA0807387', [7].Model := 'WTW4816FW2', [7].DateTime := '2/25/2021 12:29:57.14076', [8].writeIndex := 8, [8].readIndex := 8, [8].LastReadCode := 1, [8].Serial := 'CA0807388', [8].Model := 'WTW4816FW2', [8].DateTime := '2/25/2021 12:30:38.78655', [9].writeIndex := 10, [9].readIndex := 9, [9].LastReadCode := 1, [9].Serial := 'CA0807389', [9].Model := 'WTW4816FW2', [9].DateTime := '2/25/2021 12:30:51.72217', [10].writeIndex := 10, [10].readIndex := 10,
        [10].LastReadCode := 1, [10].Serial := 'CA0807390', [10].Model := 'WTW4816FW2', [10].DateTime := '2/25/2021 12:31:01.80920', [11].writeIndex := 11, [11].readIndex := 11, [11].LastReadCode := 1, [11].Serial := 'CA0807391', [11].Model := 'WTW4816FW2', [11].DateTime := '2/25/2021 12:31:11.91238', [12].writeIndex := 12, [12].readIndex := 12, [12].LastReadCode := 1, [12].Serial := 'CA0807392', [12].Model := 'WTW4816FW2', [12].DateTime := '2/25/2021 12:31:24.82835', [13].writeIndex := 13, [13].readIndex := 13, [13].LastReadCode := 1, [13].Serial := 'CA0807393', [13].Model := 'WTW4816FW2', [13].DateTime := '2/25/2021 12:31:33.33885', [14].writeIndex := 14, [14].readIndex := 14, [14].LastReadCode := 1, [14].Serial := 'CA0807394', [14].Model := 'WTW4816FW2', [14].DateTime := '2/25/2021 12:31:44.26004', [15].writeIndex := 15, [15].readIndex := 15, [15].LastReadCode := 1, [15].Serial := 'CA0807395', [15].Model := 'WTW4816FW2', [15].DateTime := '2/25/2021 12:31:55.17391', [16].writeIndex := 16, [16].readIndex := 16, [16].LastReadCode := 1, [16].Serial := 'CA0807396', [16].Model := 'WTW4816FW2', [16].DateTime := '2/25/2021 12:32:06.90771', [17].writeIndex := 17, [17].readIndex := 17, [17].LastReadCode := 1, [17].Serial := 'CA0807397', [17].Model := 'WTW4816FW2', [17].DateTime := '2/25/2021 12:32:16.96281', [18].writeIndex := 18, [18].readIndex := 18, [18].LastReadCode := 1, [18].Serial := 'CA0807398', [18].Model := 'WTW4816FW2', [18].DateTime := '2/25/2021 12:32:27.92434', [19].writeIndex := 19, [19].readIndex := 19, [19].LastReadCode := 1, [19].Serial := 'CA0807399', [19].Model := 'WTW4816FW2', [19].DateTime := '2/25/2021 12:32:38.40881', [20].writeIndex := 20, [20].readIndex := 20,
        [20].LastReadCode := 1, [20].Serial := 'CA0807400', [20].Model := 'WTW4816FW2', [20].DateTime := '2/25/2021 12:32:49.30917', [21].writeIndex := 21, [21].readIndex := 21, [21].LastReadCode := 1, [21].Serial := 'CA0807401', [21].Model := 'WTW4816FW2', [21].DateTime := '2/25/2021 12:33:00.28133', [22].writeIndex := 22, [22].readIndex := 22, [22].LastReadCode := 1, [22].Serial := 'CA0807402', [22].Model := 'WTW4816FW2', [22].DateTime := '2/25/2021 12:33:35.38591', [23].writeIndex := 23, [23].readIndex := 23, [23].LastReadCode := 1, [23].Serial := 'CA0807403', [23].Model := 'WTW4816FW2', [23].DateTime := '2/25/2021 12:33:45.88840', [24].writeIndex := 24, [24].readIndex := 24, [24].LastReadCode := 1, [24].Serial := 'CA0807404', [24].Model := 'WTW4816FW2', [24].DateTime := '2/25/2021 12:33:56.85644', [25].writeIndex := 25, [25].readIndex := 25, [25].LastReadCode := 1, [25].Serial := 'CA0807405', [25].Model := 'WTW4816FW2', [25].DateTime := '2/25/2021 12:34:07.73473', [26].writeIndex := 26, [26].readIndex := 26, [26].LastReadCode := 1, [26].Serial := 'CA0807406', [26].Model := 'WTW4816FW2', [26].DateTime := '2/25/2021 12:34:18.63707', [27].writeIndex := 27, [27].readIndex := 27, [27].LastReadCode := 1, [27].Serial := 'CA0807407', [27].Model := 'WTW4816FW2', [27].DateTime := '2/25/2021 12:34:29.95757', [28].writeIndex := 28, [28].readIndex := 28, [28].LastReadCode := 1, [28].Serial := 'CA0807408', [28].Model := 'WTW4816FW2', [28].DateTime := '2/25/2021 12:34:41.36491', [29].writeIndex := 29, [29].readIndex := 29, [29].LastReadCode := 1, [29].Serial := 'CA0807409', [29].Model := 'WTW4816FW2', [29].DateTime := '2/25/2021 12:34:52.31039', [30].writeIndex := 30, [30].readIndex := 30,
        [30].LastReadCode := 1, [30].Serial := 'CA0807410', [30].Model := 'WTW4816FW2', [30].DateTime := '2/25/2021 12:35:05.61831', [31].writeIndex := 31, [31].readIndex := 31, [31].LastReadCode := 1, [31].Serial := 'CA0807411', [31].Model := 'WTW4816FW2', [31].DateTime := '2/25/2021 12:35:14.80057', [32].writeIndex := 32, [32].readIndex := 32, [32].LastReadCode := 1, [32].Serial := 'CA0807412', [32].Model := 'WTW4816FW2', [32].DateTime := '2/25/2021 12:35:24.99536', [33].writeIndex := 33, [33].readIndex := 33, [33].LastReadCode := 1, [33].Serial := 'CA0807413', [33].Model := 'WTW4816FW2', [33].DateTime := '2/25/2021 12:35:35.89756', [34].writeIndex := 34, [34].readIndex := 34, [34].LastReadCode := 1, [34].Serial := 'CA0807414', [34].Model := 'WTW4816FW2', [34].DateTime := '2/25/2021 12:35:49.25334', [35].writeIndex := 35, [35].readIndex := 35, [35].LastReadCode := 1, [35].Serial := 'CA0807415', [35].Model := 'WTW4816FW2', [35].DateTime := '2/25/2021 12:35:57.77427', [36].writeIndex := 36, [36].readIndex := 36, [36].LastReadCode := 1, [36].Serial := 'CA0807416', [36].Model := 'WTW4816FW2', [36].DateTime := '2/25/2021 12:36:08.66572', [37].writeIndex := 37, [37].readIndex := 37, [37].LastReadCode := 1, [37].Serial := 'CA0807417', [37].Model := 'WTW4816FW2', [37].DateTime := '2/25/2021 12:36:19.57452', [38].writeIndex := 38, [38].readIndex := 38, [38].LastReadCode := 1, [38].Serial := 'CA0807418', [38].Model := 'WTW4816FW2', [38].DateTime := '2/25/2021 12:36:30.10790', [39].writeIndex := 39, [39].readIndex := 39, [39].LastReadCode := 1, [39].Serial := 'CA0807419', [39].Model := 'WTW4816FW2', [39].DateTime := '2/25/2021 12:36:40.99675', [40].writeIndex := 40, [40].readIndex := 40,
        [40].LastReadCode := 1, [40].Serial := 'CA0807420', [40].Model := 'WTW4816FW2', [40].DateTime := '2/25/2021 12:36:51.92086', [41].writeIndex := 41, [41].readIndex := 41, [41].LastReadCode := 1, [41].Serial := 'CA0807371', [41].Model := 'WTW4816FW2', [41].DateTime := '2/25/2021 12:27:03.39945', [42].writeIndex := 42, [42].readIndex := 42, [42].LastReadCode := 1, [42].Serial := 'CA0807372', [42].Model := 'WTW4816FW2', [42].DateTime := '2/25/2021 12:27:14.31229', [43].writeIndex := 43, [43].readIndex := 43, [43].LastReadCode := 1, [43].Serial := 'CA0807373', [43].Model := 'WTW4816FW2', [43].DateTime := '2/25/2021 12:27:25.22997', [44].writeIndex := 44, [44].readIndex := 44, [44].LastReadCode := 1, [44].Serial := 'CA0807374', [44].Model := 'WTW4816FW2', [44].DateTime := '2/25/2021 12:27:36.12574', [45].writeIndex := 45, [45].readIndex := 45, [45].LastReadCode := 1, [45].Serial := 'CA0807375', [45].Model := 'WTW4816FW2', [45].DateTime := '2/25/2021 12:27:46.64041', [46].writeIndex := 46, [46].readIndex := 46, [46].LastReadCode := 1, [46].Serial := 'CA0807376', [46].Model := 'WTW4816FW2', [46].DateTime := '2/25/2021 12:27:57.56194', [47].writeIndex := 47, [47].readIndex := 47, [47].LastReadCode := 1, [47].Serial := 'CA0807377', [47].Model := 'WTW4816FW2', [47].DateTime := '2/25/2021 12:28:08.50169', [48].writeIndex := 48, [48].readIndex := 48, [48].LastReadCode := 1, [48].Serial := 'CA0807378', [48].Model := 'WTW4816FW2', [48].DateTime := '2/25/2021 12:28:19.39640', [49].writeIndex := 49, [49].readIndex := 49, [49].LastReadCode := 1, [49].Serial := 'CA0807379', [49].Model := 'WTW4816FW2', [49].DateTime := '2/25/2021 12:28:30.29576');
   LN04_SNModel_CurrentRead : UDT_SN_Model := (writeIndex := 38, readIndex := 38, Serial := 'CA0807418', Model := 'WTW4816FW2', DateTime := '2/25/2021 12:36:30.10790');
   LN04_SNModel_STR40 : STRING_40[10] := ([0] := 'CA0807420', [1] := 'WTW4816FW2', [2] := '2/25/2021 12:36:55.546816');
   LN04_Standard_Shift_Break_In_Minutes : DINT := 50;
   LN04_StorageDrawer_MNT : DINT;
   LN04_Theoretical_Units_Counter : COUNTER := (PRE := 999999, ACC := 204);
   LN04_Theoretical_Units_Counter_ONS : BOOL;
   LN04_Toggle_CountSource : BOOL := 1;
   LN04_Units_for_repair : DINT := 100;
   LN04_Weekly_Schedule : UDT_Weekly_Schedule := (Monday._1st_Shift_Avail := 1, Monday._1st_Shift_Start := '2023-05-08 05:00', Monday._1st_Shift_End := '2023-05-08 13:30', Monday._2nd_Shift_Start := '2023-05-08 16:45', Monday._2nd_Shift_End := '2023-05-08 23:55', Monday._3rd_Shift_Start := '2023-05-08 04:50', Monday._3rd_Shift_End := '2023-05-08 04:55', Monday.S1_Scheduled := 425, Tuesday._1st_Shift_Avail := 1, Tuesday._1st_Shift_Start := '2023-05-09 05:00', Tuesday._1st_Shift_End := '2023-05-09 15:30', Tuesday._2nd_Shift_Start := '2023-05-09 16:45', Tuesday._2nd_Shift_End := '2023-05-09 23:55', Tuesday._3rd_Shift_Start := '2023-05-09 04:50', Tuesday._3rd_Shift_End := '2023-05-09 04:55', Tuesday.S1_Scheduled := 527, Wednesday._1st_Shift_Avail := 1, Wednesday._1st_Shift_Start := '2023-05-10 05:00', Wednesday._1st_Shift_End := '2023-05-10 15:30', Wednesday._2nd_Shift_Start := '2023-05-10 16:45', Wednesday._2nd_Shift_End := '2023-05-10 23:55', Wednesday._3rd_Shift_Start := '2023-05-10 04:50', Wednesday._3rd_Shift_End := '2023-05-10 04:55', Wednesday.S1_Scheduled := 527, Thursday._1st_Shift_Avail := 1, Thursday._1st_Shift_Start := '2023-05-11 05:00', Thursday._1st_Shift_End := '2023-05-11 13:30', Thursday._2nd_Shift_Start := '2023-05-11 16:45', Thursday._2nd_Shift_End := '2023-05-11 23:55', Thursday._3rd_Shift_Start := '2023-05-11 04:50', Thursday._3rd_Shift_End := '2023-05-11 04:55', Thursday.S1_Scheduled := 425, Friday._1st_Shift_Avail := 1, Friday._1st_Shift_Start := '2023-05-12 05:00', Friday._1st_Shift_End := '2023-05-12 13:30', Friday._2nd_Shift_Start := '2023-05-12 16:45', Friday._2nd_Shift_End := '2023-05-12 23:55', Friday._3rd_Shift_Start := '2023-05-12 04:50', Friday._3rd_Shift_End := '2023-05-12 04:55', Friday.S1_Scheduled := 425, Saturday._1st_Shift_Start := '2023-05-13 05:00', Saturday._1st_Shift_End := '2023-05-13 13:30', Saturday._2nd_Shift_Start := '2023-05-13 16:45', Saturday._2nd_Shift_End := '2023-05-13 23:55', Saturday._3rd_Shift_Start := '2023-05-13 04:50', Saturday._3rd_Shift_End := '2023-05-13 04:55', Sunday._1st_Shift_Start := '2023-05-14 05:00', Sunday._1st_Shift_End := '2023-05-14 13:30', Sunday._2nd_Shift_Start := '2023-05-14 16:45', Sunday._2nd_Shift_End := '2023-05-14 23:55', Sunday._3rd_Shift_Start := '2023-05-14 04:50', Sunday._3rd_Shift_End := '2023-05-14 04:55');
   LN04_Wiring_MNT : DINT;
   LN04EAM01 : DINT;
   LN04EAM02 : DINT;
   LN04ECM01 : DINT;
   LN04ECM02 : DINT;
   LN04ECM03 : DINT;
   LN04ECM04 : DINT;
   LN04ECM05 : DINT;
   LN04EDM01 : DINT;
   LN04EDM04 : DINT;
   LN04EDM06 : DINT;
   LN04EDM07 : DINT;
   LN04EDM08 : DINT;
   LN04EEM01 : DINT;
   LN04EEM02 : DINT;
   LN04EEM03 : DINT;
   LN04EES01 : DINT;
   LN04EES02 : DINT;
   LN04EES03 : DINT;
   LN04EES04 : DINT;
   LN04EFM03 : DINT;
   LN04EFS04 : DINT;
   LN04EFS05 : DINT;
   LN04EGM01 : DINT;
   LN04EGM04 : DINT;
   LN04EGS01 : DINT;
   LN04EGS02 : DINT;
   LN04EGS03 : DINT;
   LN04EHM01 : DINT;
   LN04EHM02 : DINT;
   LN04EHM03 : DINT;
   LN04EHM04 : DINT;
   LN04EHM05 : DINT;
   LN04EHM06 : DINT;
   LN04EHM07 : DINT;
   LN04EHM08 : DINT;
   LN04EJM02 : DINT;
   LN04EJM03 : DINT;
   LN04EKM01 : DINT;
   LN04EKM02 : DINT;
   LN04EKM03 : DINT;
   LN04ELM01 : DINT;
   LN04ELM02 : DINT;
   LN04ELM03 : DINT;
   LN04ELM04 : DINT;
   LN04ELM05 : DINT;
   LN04EMM01 : DINT;
   LN04EMM02 : DINT;
   LN04EMM03 : DINT;
   LN04EMM04 : DINT;
   LN04NAS01 : DINT;
   LN04NAS02 : DINT;
   LN04NAS03 : DINT;
   LN04NBS01 : DINT;
   LN04NBS02 : DINT;
   LN04NNM02 : DINT;
   LN04SAS01 : DINT;
   LN04SAS02 : DINT;
   LN04SAS03 : DINT;
   LN04SBS01 : DINT;
   LN04SBS03 : DINT;
   LN04SDS01 : DINT;
   LN04SFS03 : DINT;
   LN04SKS05 : DINT;
   LN04SLS01 : DINT;
   LN04SLS02 : DINT;
   LN04SLS03 : DINT;
   LN04SMM02 : DINT;
   LN04SMN02 : DINT := 16;
   LN04SNM02 : DINT;
   LN04WAM01 : DINT;
   LN04WBM01 : DINT;
   LN04WBM02 : DINT;
   LN04WBM03 : DINT;
   LN04WBM04 : DINT;
   LN04WCM01 : DINT;
   LN04WCM02 : DINT;
   LN04WCM03 : DINT;
   LN04WCM04 : DINT;
   LN04WCM05 : DINT;
   LN04WCM06 : DINT;
   LN04WCS01 : DINT;
   LN04WDM01 : DINT;
   LN04WDM02 : DINT;
   LN04WDM03 : DINT;
   LN04WDM04 : DINT;
   LN04WDM05 : DINT;
   LN04WEM01 : DINT;
   LN04WEM02 : DINT;
   LN04WEM03 : DINT;
   LN04WFM01 : DINT;
   LN04WFM02 : DINT;
   LN04WFM03 : DINT;
   LN04WFM04 : DINT;
   LN04WFM05 : DINT;
   LN04WFS01 : DINT;
   LN04WFS02 : DINT;
   LN04WGM01 : DINT;
   LN04WGM02 : DINT;
   LN04WGM03 : DINT;
   LN04WGM04 : DINT;
   LN04WGM05 : DINT;
   LN04WHM08 : DINT;
   LN04WHM09 : DINT;
   LN04WJM01 : DINT;
   LN04WJM02 : DINT;
   LN04WJM03 : DINT;
   LN04WJS01 : DINT;
   LN04WJS02 : DINT;
   LN04WJS03 : DINT;
   LN04WKM01 : DINT;
   LN04WKM02 : DINT;
   LN04WKM03 : DINT;
   LN04WKS01 : DINT;
   LN04WKS02 : DINT;
   LN04WKS03 : DINT;
   LN04WKS04 : DINT;
   LN04WLM01 : DINT;
   LN04WLM06 : DINT;
   LN04WLM07 : DINT;
   LN04WMM01 : DINT;
   LN04WMM02 : DINT;
   LN04WMM03 : DINT;
   LN04WMM04 : DINT;
   LN04WNM01 : DINT;
   LN04ZMN01 : DINT;
   LN04ZMN02 : DINT;
   LN04ZMN03 : DINT;
   LN04ZMN04 : DINT;
   LN04ZMS01 : DINT;
   LN04ZMS02 : DINT;
   LN04ZMS03 : DINT;
   LN04ZMS04 : DINT;
   mlc_test21 : BOOL;
   msg192_reset_timer : TIMER := (PRE := 3000);
   null : STRING;
   Previous_Shift_Count : DINT;
   R2_Data : R1_Lines_Status_to_R2 := (LN02.Count := 1734, LN03.Count := 2416, LN03.Break_Active := 1, LN04.Active_Shift := 1, LN04.Count := 1866, LN07.Active_Shift := 1, LN07.DT_Active := 1);
   scc : CONTROL := (LEN := 60, POS := 59);
   Shift_count_history : DINT[62] := ([1] := 1, [2] := 1, [5] := 1, [6] := 1, [12] := 1, [13] := 1, [18] := 1, [19] := 1, [26] := 1, [30] := 1, [31] := 1, [33] := 1, [39] := 1, [41] := 1, [42] := 1, [46] := 1, [47] := 1, [48] := 1, [57] := 1);
   Shift_reset_timer : TIMER := (PRE := 2000);
   STR_Null : STRING;
   test : BOOL;
   Test_APC : DINT := 18;
   Test_Bit : DINT;
   TEST_CTR_APC1 : COUNTER := (PRE := 99999999, ACC := 771);
   Test_Result : DINT;
   test_snn : BOOL;
   TestDateTime : DINT;
   TMR_COMMS : TIMER := (PRE := 10000, EN := 1, DN := 1);
END_VAR
